LIN {X 0,Y 227.274,Z 763.314,A -85,B 0,C 180,E1 -20014.895,E2 -20014.895} C_VEL
LIN {X 0,Y 226.122,Z 765.679,A -85,B 0,C 180,E1 -20018.434,E2 -20018.434} C_VEL
LIN {X 0,Y 225.536,Z 766.463,A -85,B 0,C 180,E1 -20021.593,E2 -20021.593} C_VEL
LIN {X 0,Y 225.305,Z 766.2,A -85,B 0,C 180,E1 -20024.155,E2 -20024.155} C_VEL
LIN {X 0,Y 225.347,Z 765.158,A -85,B 0,C 180,E1 -20026.675,E2 -20026.675} C_VEL
LIN {X 0,Y 225.598,Z 763.327,A -85,B 0,C 180,E1 -20029.14,E2 -20029.14} C_VEL
LIN {X 0,Y 225.943,Z 760.772,A -85,B 0,C 180,E1 -20031.529,E2 -20031.529} C_VEL
LIN {X 0,Y 226.464,Z 757.485,A -85,B 0,C 180,E1 -20033.868,E2 -20033.868} C_VEL
LIN {X 0,Y 227.318,Z 752.537,A -85,B 0,C 180,E1 -20036.591,E2 -20036.591} C_VEL
LIN {X 0,Y 228.588,Z 745.96,A -85,B 0,C 180,E1 -20039.415,E2 -20039.415} C_VEL
LIN {X 0,Y 230.085,Z 738.559,A -85,B 0,C 180,E1 -20041.941,E2 -20041.941} C_VEL
LIN {X 0,Y 231.914,Z 729.456,A -85,B 0,C 180,E1 -20044.415,E2 -20044.415} C_VEL
LIN {X 0,Y 233.849,Z 719.737,A -85,B 0,C 180,E1 -20046.533,E2 -20046.533} C_VEL
LIN {X 0,Y 235.817,Z 708.858,A -85,B 0,C 180,E1 -20048.434,E2 -20048.434} C_VEL
LIN {X 0,Y 236.209,Z 705.915,A -85,B 0,C 180,E1 -20048.878,E2 -20048.878} C_VEL
LIN {X 0,Y 234.743,Z 695.22,A -85,B 0,C 180,E1 -20050.544,E2 -20050.544} C_VEL
LIN {X 0,Y 232.764,Z 684.343,A -85,B 0,C 180,E1 -20051.988,E2 -20051.988} C_VEL
LIN {X 0,Y 229.693,Z 671.184,A -85,B 0,C 180,E1 -20053.426,E2 -20053.426} C_VEL
LIN {X 0,Y 227.253,Z 661.617,A -85,B 0,C 180,E1 -20054.299,E2 -20054.299} C_VEL
LIN {X 0,Y 227.825,Z 657.568,A -85,B 0,C 180,E1 -20059.333,E2 -20059.333} C_VEL
LIN {X 0,Y 228.196,Z 656.059,A -85,B 0,C 180,E1 -20061.364,E2 -20061.364} C_VEL
LIN {X 0,Y 228.175,Z 656.064,A -85,B 0,C 180,E1 -20064.697,E2 -20064.697} C_VEL
LIN {X 0,Y 228.557,Z 656.012,A -85,B 0,C 180,E1 -20068.237,E2 -20068.237} C_VEL
LIN {X 0,Y 228.556,Z 656.01,A -85,B 0,C 180,E1 -20071.761,E2 -20071.761} C_VEL
LIN {X 0,Y 228.191,Z 656.057,A -85,B 0,C 180,E1 -20077.076,E2 -20077.076} C_VEL
LIN {X 0,Y 227.745,Z 656.119,A -85,B 0,C 180,E1 -20081.119,E2 -20081.119} C_VEL
LIN {X 0,Y 227.625,Z 656.245,A -85,B 0,C 180,E1 -20081.576,E2 -20081.576} C_VEL
LIN {X 0,Y 227.143,Z 659.782,A -85,B 0,C 180,E1 -20084.788,E2 -20084.788} C_VEL
LIN {X 0,Y 230.876,Z 674.703,A -85,B 0,C 180,E1 -20086.162,E2 -20086.162} C_VEL
LIN {X 0,Y 233.355,Z 686.703,A -85,B 0,C 180,E1 -20087.527,E2 -20087.527} C_VEL
LIN {X 0,Y 235.304,Z 698.674,A -85,B 0,C 180,E1 -20089.18,E2 -20089.18} C_VEL
LIN {X 0,Y 236.095,Z 705.463,A -85,B 0,C 180,E1 -20090.245,E2 -20090.245} C_VEL
LIN {X 0,Y 234.36,Z 715.909,A -85,B 0,C 180,E1 -20091.953,E2 -20091.953} C_VEL
LIN {X 0,Y 232.354,Z 726.447,A -85,B 0,C 180,E1 -20094.099,E2 -20094.099} C_VEL
LIN {X 0,Y 230.69,Z 734.831,A -85,B 0,C 180,E1 -20096.214,E2 -20096.214} C_VEL
LIN {X 0,Y 228.896,Z 743.456,A -85,B 0,C 180,E1 -20098.94,E2 -20098.94} C_VEL
LIN {X 0,Y 227.645,Z 750.251,A -85,B 0,C 180,E1 -20101.656,E2 -20101.656} C_VEL
LIN {X 0,Y 226.787,Z 754.751,A -85,B 0,C 180,E1 -20103.903,E2 -20103.903} C_VEL
LIN {X 0,Y 226.156,Z 758.446,A -85,B 0,C 180,E1 -20106.187,E2 -20106.187} C_VEL
LIN {X 0,Y 225.597,Z 761.739,A -85,B 0,C 180,E1 -20108.847,E2 -20108.847} C_VEL
LIN {X 0,Y 225.241,Z 764.045,A -85,B 0,C 180,E1 -20111.509,E2 -20111.509} C_VEL
LIN {X 0,Y 225.231,Z 765.419,A -85,B 0,C 180,E1 -20114.136,E2 -20114.136} C_VEL
LIN {X 0,Y 225.354,Z 765.922,A -85,B 0,C 180,E1 -20116.677,E2 -20116.677} C_VEL
LIN {X 0,Y 225.717,Z 765.607,A -85,B 0,C 180,E1 -20119.166,E2 -20119.166} C_VEL
LIN {X 0,Y 226.268,Z 764.569,A -85,B 0,C 180,E1 -20121.595,E2 -20121.595} C_VEL
LIN {X 0,Y 227.147,Z 762.813,A -85,B 0,C 180,E1 -20123.994,E2 -20123.994} C_VEL
LIN {X 0,Y 228.834,Z 758.808,A -85,B 0,C 180,E1 -20127.489,E2 -20127.489} C_VEL
LIN {X 0,Y 230.384,Z 754.929,A -85,B 0,C 180,E1 -20129.916,E2 -20129.916} C_VEL
LIN {X 0,Y 232.388,Z 749.966,A -85,B 0,C 180,E1 -20132.35,E2 -20132.35} C_VEL
LIN {X 0,Y 234.755,Z 743.842,A -85,B 0,C 180,E1 -20134.744,E2 -20134.744} C_VEL
LIN {X 0,Y 237.51,Z 736.342,A -85,B 0,C 180,E1 -20137.093,E2 -20137.093} C_VEL
LIN {X 0,Y 240.476,Z 727.629,A -85,B 0,C 180,E1 -20139.26,E2 -20139.26} C_VEL
LIN {X 0,Y 243.611,Z 717.397,A -85,B 0,C 180,E1 -20141.28,E2 -20141.28} C_VEL
LIN {X 0,Y 244.299,Z 713.897,A -85,B 0,C 180,E1 -20141.926,E2 -20141.926} C_VEL
LIN {X 0,Y 243.791,Z 704.371,A -85,B 0,C 180,E1 -20143.891,E2 -20143.891} C_VEL
LIN {X 0,Y 242.005,Z 693.516,A -85,B 0,C 180,E1 -20146.031,E2 -20146.031} C_VEL
LIN {X 0,Y 239.114,Z 682.956,A -85,B 0,C 180,E1 -20148.127,E2 -20148.127} C_VEL
LIN {X 0,Y 235.916,Z 674.484,A -85,B 0,C 180,E1 -20149.85,E2 -20149.85} C_VEL
LIN {X 0,Y 233.629,Z 669.665,A -85,B 0,C 180,E1 -20150.93,E2 -20150.93} C_VEL
LIN {X 0,Y 231.756,Z 665.99,A -85,B 0,C 180,E1 -20151.773,E2 -20151.773} C_VEL
LIN {X 0,Y 229.771,Z 662.892,A -85,B 0,C 180,E1 -20152.586,E2 -20152.586} C_VEL
LIN {X 0,Y 229.263,Z 661.334,A -85,B 0,C 180,E1 -20152.901,E2 -20152.901} C_VEL
LIN {X 0,Y 228.776,Z 657.181,A -85,B 0,C 180,E1 -20158.24,E2 -20158.24} C_VEL
LIN {X 0,Y 228.623,Z 656.007,A -85,B 0,C 180,E1 -20160,E2 -20160} C_VEL
LIN {X 0,Y 228.553,Z 656.016,A -85,B 0,C 180,E1 -20161.762,E2 -20161.762} C_VEL
LIN {X 0,Y 228.355,Z 656.04,A -85,B 0,C 180,E1 -20167.071,E2 -20167.071} C_VEL
LIN {X 0,Y 228.169,Z 656.065,A -85,B 0,C 180,E1 -20170.65,E2 -20170.65} C_VEL
LIN {X 0,Y 228.055,Z 656.076,A -85,B 0,C 180,E1 -20176.102,E2 -20176.102} C_VEL
LIN {X 0,Y 227.94,Z 656.092,A -85,B 0,C 180,E1 -20179.826,E2 -20179.826} C_VEL
LIN {X 0,Y 227.911,Z 656.092,A -85,B 0,C 180,E1 -20183.633,E2 -20183.633} C_VEL
LIN {X 0,Y 227.883,Z 656.1,A -85,B 0,C 180,E1 -20187.555,E2 -20187.555} C_VEL
LIN {X 0,Y 227.869,Z 656.1,A -85,B 0,C 180,E1 -20191.622,E2 -20191.622} C_VEL
LIN {X 0,Y 227.88,Z 656.097,A -85,B 0,C 180,E1 -20195.872,E2 -20195.872} C_VEL
LIN {X 0,Y 227.829,Z 656.101,A -85,B 0,C 180,E1 -20198.548,E2 -20198.548} C_VEL
LIN {X 0,Y 227.18,Z 656.345,A -85,B 0,C 180,E1 -20200.022,E2 -20200.022} C_VEL
LIN {X 0,Y 225.688,Z 657.012,A -85,B 0,C 180,E1 -20201.468,E2 -20201.468} C_VEL
LIN {X 0,Y 222.387,Z 659.357,A -85,B 0,C 180,E1 -20204.352,E2 -20204.352} C_VEL
LIN {X 0,Y 221.675,Z 660.931,A -85,B 0,C 180,E1 -20205.825,E2 -20205.825} C_VEL
LIN {X 0,Y 221.72,Z 661.5,A -85,B 0,C 180,E1 -20206.317,E2 -20206.317} C_VEL
LIN {X 0,Y 222.548,Z 665.01,A -85,B 0,C 180,E1 -20209.016,E2 -20209.016} C_VEL
LIN {X 0,Y 225.07,Z 669.34,A -85,B 0,C 180,E1 -20210.166,E2 -20210.166} C_VEL
LIN {X 0,Y 226.351,Z 672.017,A -85,B 0,C 180,E1 -20210.777,E2 -20210.777} C_VEL
LIN {X 0,Y 228.189,Z 675.676,A -85,B 0,C 180,E1 -20211.635,E2 -20211.635} C_VEL
LIN {X 0,Y 231.062,Z 684.216,A -85,B 0,C 180,E1 -20213.274,E2 -20213.274} C_VEL
LIN {X 0,Y 233.784,Z 695.583,A -85,B 0,C 180,E1 -20215.343,E2 -20215.343} C_VEL
LIN {X 0,Y 235.256,Z 705.746,A -85,B 0,C 180,E1 -20217.171,E2 -20217.171} C_VEL
LIN {X 0,Y 235.869,Z 716.507,A -85,B 0,C 180,E1 -20219.195,E2 -20219.195} C_VEL
LIN {X 0,Y 235.472,Z 726.605,A -85,B 0,C 180,E1 -20221.221,E2 -20221.221} C_VEL
LIN {X 0,Y 234.448,Z 733.894,A -85,B 0,C 180,E1 -20222.798,E2 -20222.798} C_VEL
LIN {X 0,Y 231.402,Z 742.92,A -85,B 0,C 180,E1 -20224.838,E2 -20224.838} C_VEL
LIN {X 0,Y 228.129,Z 751.752,A -85,B 0,C 180,E1 -20227.353,E2 -20227.353} C_VEL
LIN {X 0,Y 225.399,Z 758.948,A -85,B 0,C 180,E1 -20229.942,E2 -20229.942} C_VEL
LIN {X 0,Y 223.2,Z 764.764,A -85,B 0,C 180,E1 -20232.595,E2 -20232.595} C_VEL
LIN {X 0,Y 221.234,Z 769.387,A -85,B 0,C 180,E1 -20235.278,E2 -20235.278} C_VEL
LIN {X 0,Y 219.983,Z 772.932,A -85,B 0,C 180,E1 -20238.016,E2 -20238.016} C_VEL
LIN {X 0,Y 219.133,Z 775.505,A -85,B 0,C 180,E1 -20240.773,E2 -20240.773} C_VEL
LIN {X 0,Y 218.765,Z 776.719,A -85,B 0,C 180,E1 -20242.618,E2 -20242.618} C_VEL
LIN {X 0,Y 218.557,Z 777.78,A -85,B 0,C 180,E1 -20245.45,E2 -20245.45} C_VEL
LIN {X 0,Y 218.602,Z 778.042,A -85,B 0,C 180,E1 -20248.158,E2 -20248.158} C_VEL
LIN {X 0,Y 218.67,Z 778.897,A -85,B 0,C 180,E1 -20250.001,E2 -20250.001} C_VEL
LIN {X 0,Y 218.561,Z 779.313,A -85,B 0,C 180,E1 -20251.843,E2 -20251.843} C_VEL
LIN {X 0,Y 218.597,Z 778.94,A -85,B 0,C 180,E1 -20255.536,E2 -20255.536} C_VEL
LIN {X 0,Y 218.797,Z 778.178,A -85,B 0,C 180,E1 -20257.383,E2 -20257.383} C_VEL
LIN {X 0,Y 219.145,Z 777.013,A -85,B 0,C 180,E1 -20259.228,E2 -20259.228} C_VEL
LIN {X 0,Y 220.412,Z 773.422,A -85,B 0,C 180,E1 -20262.898,E2 -20262.898} C_VEL
LIN {X 0,Y 221.86,Z 769.607,A -85,B 0,C 180,E1 -20265.621,E2 -20265.621} C_VEL
LIN {X 0,Y 223.99,Z 764.713,A -85,B 0,C 180,E1 -20268.287,E2 -20268.287} C_VEL
LIN {X 0,Y 226.381,Z 758.62,A -85,B 0,C 180,E1 -20270.918,E2 -20270.918} C_VEL
LIN {X 0,Y 229.184,Z 751.13,A -85,B 0,C 180,E1 -20273.494,E2 -20273.494} C_VEL
LIN {X 0,Y 232.086,Z 743.584,A -85,B 0,C 180,E1 -20275.564,E2 -20275.564} C_VEL
LIN {X 0,Y 235.421,Z 733.539,A -85,B 0,C 180,E1 -20277.805,E2 -20277.805} C_VEL
LIN {X 0,Y 236.271,Z 724.664,A -85,B 0,C 180,E1 -20279.735,E2 -20279.735} C_VEL
LIN {X 0,Y 236.179,Z 715.261,A -85,B 0,C 180,E1 -20281.657,E2 -20281.657} C_VEL
LIN {X 0,Y 235.121,Z 705.444,A -85,B 0,C 180,E1 -20283.616,E2 -20283.616} C_VEL
LIN {X 0,Y 233.152,Z 695.824,A -85,B 0,C 180,E1 -20285.524,E2 -20285.524} C_VEL
LIN {X 0,Y 229.982,Z 685.655,A -85,B 0,C 180,E1 -20287.675,E2 -20287.675} C_VEL
LIN {X 0,Y 228.05,Z 681.227,A -85,B 0,C 180,E1 -20288.719,E2 -20288.719} C_VEL
LIN {X 0,Y 226.282,Z 677.271,A -85,B 0,C 180,E1 -20289.681,E2 -20289.681} C_VEL
LIN {X 0,Y 223.674,Z 673.089,A -85,B 0,C 180,E1 -20290.949,E2 -20290.949} C_VEL
LIN {X 0,Y 223.107,Z 671.11,A -85,B 0,C 180,E1 -20291.351,E2 -20291.351} C_VEL
LIN {X 0,Y 222.919,Z 669.385,A -85,B 0,C 180,E1 -20293.916,E2 -20293.916} C_VEL
LIN {X 0,Y 222.468,Z 666.7,A -85,B 0,C 180,E1 -20298.439,E2 -20298.439} C_VEL
LIN {X 0,Y 222.139,Z 664.407,A -85,B 0,C 180,E1 -20303.05,E2 -20303.05} C_VEL
LIN {X 0,Y 221.847,Z 662.686,A -85,B 0,C 180,E1 -20307.415,E2 -20307.415} C_VEL
LIN {X 0,Y 221.656,Z 661.448,A -85,B 0,C 180,E1 -20311.601,E2 -20311.601} C_VEL
LIN {X 0,Y 221.53,Z 660.632,A -85,B 0,C 180,E1 -20315.643,E2 -20315.643} C_VEL
LIN {X 0,Y 221.475,Z 660.194,A -85,B 0,C 180,E1 -20319.57,E2 -20319.57} C_VEL
LIN {X 0,Y 221.582,Z 660.074,A -85,B 0,C 180,E1 -20323.414,E2 -20323.414} C_VEL
LIN {X 0,Y 221.654,Z 660.293,A -85,B 0,C 180,E1 -20327.176,E2 -20327.176} C_VEL
LIN {X 0,Y 221.899,Z 660.774,A -85,B 0,C 180,E1 -20330.888,E2 -20330.888} C_VEL
LIN {X 0,Y 222.014,Z 661.565,A -85,B 0,C 180,E1 -20334.551,E2 -20334.551} C_VEL
LIN {X 0,Y 222.44,Z 662.548,A -85,B 0,C 180,E1 -20338.19,E2 -20338.19} C_VEL
LIN {X 0,Y 222.644,Z 663.12,A -85,B 0,C 180,E1 -20340,E2 -20340} C_VEL
LIN {X 0,Y 222.533,Z 664.557,A -85,B 0,C 180,E1 -20343.565,E2 -20343.565} C_VEL
LIN {X 0,Y 223.667,Z 667.608,A -85,B 0,C 180,E1 -20344.281,E2 -20344.281} C_VEL
LIN {X 0,Y 225.776,Z 670.33,A -85,B 0,C 180,E1 -20345.268,E2 -20345.268} C_VEL
LIN {X 0,Y 227.849,Z 674.14,A -85,B 0,C 180,E1 -20346.364,E2 -20346.364} C_VEL
LIN {X 0,Y 231.352,Z 681.619,A -85,B 0,C 180,E1 -20348.297,E2 -20348.297} C_VEL
LIN {X 0,Y 234.93,Z 692.21,A -85,B 0,C 180,E1 -20350.775,E2 -20350.775} C_VEL
LIN {X 0,Y 237.082,Z 701.465,A -85,B 0,C 180,E1 -20352.846,E2 -20352.846} C_VEL
LIN {X 0,Y 238.267,Z 710.869,A -85,B 0,C 180,E1 -20354.957,E2 -20354.957} C_VEL
LIN {X 0,Y 238.439,Z 717.51,A -85,B 0,C 180,E1 -20356.481,E2 -20356.481} C_VEL
LIN {X 0,Y 235.322,Z 727.408,A -85,B 0,C 180,E1 -20358.464,E2 -20358.464} C_VEL
LIN {X 0,Y 232.446,Z 735.279,A -85,B 0,C 180,E1 -20360.398,E2 -20360.398} C_VEL
LIN {X 0,Y 229.065,Z 743.764,A -85,B 0,C 180,E1 -20363.009,E2 -20363.009} C_VEL
LIN {X 0,Y 226.156,Z 750.779,A -85,B 0,C 180,E1 -20365.789,E2 -20365.789} C_VEL
LIN {X 0,Y 223.837,Z 756.029,A -85,B 0,C 180,E1 -20368.46,E2 -20368.46} C_VEL
LIN {X 0,Y 221.945,Z 760.206,A -85,B 0,C 180,E1 -20371.243,E2 -20371.243} C_VEL
LIN {X 0,Y 220.515,Z 763.269,A -85,B 0,C 180,E1 -20374.04,E2 -20374.04} C_VEL
LIN {X 0,Y 219.266,Z 765.708,A -85,B 0,C 180,E1 -20377.517,E2 -20377.517} C_VEL
LIN {X 0,Y 218.668,Z 766.536,A -85,B 0,C 180,E1 -20380.001,E2 -20380.001} C_VEL
LIN {X 0,Y 218.324,Z 766.658,A -85,B 0,C 180,E1 -20382.532,E2 -20382.532} C_VEL
LIN {X 0,Y 218.212,Z 766.033,A -85,B 0,C 180,E1 -20385.118,E2 -20385.118} C_VEL
LIN {X 0,Y 218.347,Z 764.572,A -85,B 0,C 180,E1 -20387.758,E2 -20387.758} C_VEL
LIN {X 0,Y 218.651,Z 762.155,A -85,B 0,C 180,E1 -20390.482,E2 -20390.482} C_VEL
LIN {X 0,Y 219.182,Z 758.661,A -85,B 0,C 180,E1 -20393.285,E2 -20393.285} C_VEL
LIN {X 0,Y 220.04,Z 753.926,A -85,B 0,C 180,E1 -20396.143,E2 -20396.143} C_VEL
LIN {X 0,Y 221.243,Z 747.658,A -85,B 0,C 180,E1 -20399.058,E2 -20399.058} C_VEL
LIN {X 0,Y 222.923,Z 739.639,A -85,B 0,C 180,E1 -20401.976,E2 -20401.976} C_VEL
LIN {X 0,Y 224.749,Z 730.916,A -85,B 0,C 180,E1 -20404.5,E2 -20404.5} C_VEL
LIN {X 0,Y 226.878,Z 720.727,A -85,B 0,C 180,E1 -20406.83,E2 -20406.83} C_VEL
LIN {X 0,Y 228.961,Z 709.618,A -85,B 0,C 180,E1 -20408.858,E2 -20408.858} C_VEL
LIN {X 0,Y 229.303,Z 706.457,A -85,B 0,C 180,E1 -20409.361,E2 -20409.361} C_VEL
LIN {X 0,Y 227.826,Z 695.656,A -85,B 0,C 180,E1 -20411.1,E2 -20411.1} C_VEL
LIN {X 0,Y 225.656,Z 683.949,A -85,B 0,C 180,E1 -20412.7,E2 -20412.7} C_VEL
LIN {X 0,Y 222.676,Z 671.185,A -85,B 0,C 180,E1 -20414.144,E2 -20414.144} C_VEL
LIN {X 0,Y 220.233,Z 661.821,A -85,B 0,C 180,E1 -20415.031,E2 -20415.031} C_VEL
LIN {X 0,Y 221.106,Z 657.109,A -85,B 0,C 180,E1 -20421.085,E2 -20421.085} C_VEL
LIN {X 0,Y 221.219,Z 656.926,A -85,B 0,C 180,E1 -20422.699,E2 -20422.699} C_VEL
LIN {X 0,Y 221.515,Z 656.889,A -85,B 0,C 180,E1 -20428.181,E2 -20428.181} C_VEL
LIN {X 0,Y 221.514,Z 656.887,A -85,B 0,C 180,E1 -20431.817,E2 -20431.817} C_VEL
LIN {X 0,Y 221.117,Z 656.936,A -85,B 0,C 180,E1 -20437.303,E2 -20437.303} C_VEL
LIN {X 0,Y 220.707,Z 656.995,A -85,B 0,C 180,E1 -20441.014,E2 -20441.014} C_VEL
LIN {X 0,Y 220.6,Z 657.157,A -85,B 0,C 180,E1 -20441.484,E2 -20441.484} C_VEL
LIN {X 0,Y 220.152,Z 660.141,A -85,B 0,C 180,E1 -20444.087,E2 -20444.087} C_VEL
LIN {X 0,Y 223.775,Z 674.308,A -85,B 0,C 180,E1 -20445.424,E2 -20445.424} C_VEL
LIN {X 0,Y 226.417,Z 686.993,A -85,B 0,C 180,E1 -20446.917,E2 -20446.917} C_VEL
LIN {X 0,Y 228.362,Z 698.959,A -85,B 0,C 180,E1 -20448.62,E2 -20448.62} C_VEL
LIN {X 0,Y 229.151,Z 707.109,A -85,B 0,C 180,E1 -20449.949,E2 -20449.949} C_VEL
LIN {X 0,Y 227,Z 718.98,A -85,B 0,C 180,E1 -20452.023,E2 -20452.023} C_VEL
LIN {X 0,Y 224.908,Z 729.43,A -85,B 0,C 180,E1 -20454.366,E2 -20454.366} C_VEL
LIN {X 0,Y 223.155,Z 737.692,A -85,B 0,C 180,E1 -20456.665,E2 -20456.665} C_VEL
LIN {X 0,Y 221.495,Z 745.734,A -85,B 0,C 180,E1 -20459.459,E2 -20459.459} C_VEL
LIN {X 0,Y 220.225,Z 752.202,A -85,B 0,C 180,E1 -20462.329,E2 -20462.329} C_VEL
LIN {X 0,Y 219.303,Z 757.291,A -85,B 0,C 180,E1 -20465.228,E2 -20465.228} C_VEL
LIN {X 0,Y 218.712,Z 760.533,A -85,B 0,C 180,E1 -20467.627,E2 -20467.627} C_VEL
LIN {X 0,Y 218.292,Z 763.053,A -85,B 0,C 180,E1 -20470.082,E2 -20470.082} C_VEL
LIN {X 0,Y 218.126,Z 764.828,A -85,B 0,C 180,E1 -20472.579,E2 -20472.579} C_VEL
LIN {X 0,Y 218.143,Z 765.841,A -85,B 0,C 180,E1 -20475.135,E2 -20475.135} C_VEL
LIN {X 0,Y 218.379,Z 766.099,A -85,B 0,C 180,E1 -20477.747,E2 -20477.747} C_VEL
LIN {X 0,Y 218.862,Z 765.548,A -85,B 0,C 180,E1 -20480.413,E2 -20480.413} C_VEL
LIN {X 0,Y 219.68,Z 764.139,A -85,B 0,C 180,E1 -20483.109,E2 -20483.109} C_VEL
LIN {X 0,Y 220.824,Z 761.805,A -85,B 0,C 180,E1 -20485.839,E2 -20485.839} C_VEL
LIN {X 0,Y 222.359,Z 758.453,A -85,B 0,C 180,E1 -20488.579,E2 -20488.579} C_VEL
LIN {X 0,Y 224.29,Z 753.948,A -85,B 0,C 180,E1 -20491.324,E2 -20491.324} C_VEL
LIN {X 0,Y 227.066,Z 747.424,A -85,B 0,C 180,E1 -20494.321,E2 -20494.321} C_VEL
LIN {X 0,Y 229.652,Z 740.988,A -85,B 0,C 180,E1 -20496.645,E2 -20496.645} C_VEL
LIN {X 0,Y 233.016,Z 732.041,A -85,B 0,C 180,E1 -20499.224,E2 -20499.224} C_VEL
LIN {X 0,Y 236.323,Z 722.47,A -85,B 0,C 180,E1 -20501.367,E2 -20501.367} C_VEL
LIN {X 0,Y 238.115,Z 716.596,A -85,B 0,C 180,E1 -20502.479,E2 -20502.479} C_VEL
LIN {X 0,Y 238.001,Z 708.977,A -85,B 0,C 180,E1 -20504.148,E2 -20504.148} C_VEL
LIN {X 0,Y 236.866,Z 699.006,A -85,B 0,C 180,E1 -20506.269,E2 -20506.269} C_VEL
LIN {X 0,Y 234.397,Z 688.259,A -85,B 0,C 180,E1 -20508.549,E2 -20508.549} C_VEL
LIN {X 0,Y 231.629,Z 679.76,A -85,B 0,C 180,E1 -20510.393,E2 -20510.393} C_VEL
LIN {X 0,Y 227.968,Z 671.519,A -85,B 0,C 180,E1 -20512.36,E2 -20512.36} C_VEL
LIN {X 0,Y 225.794,Z 667.824,A -85,B 0,C 180,E1 -20513.403,E2 -20513.403} C_VEL
LIN {X 0,Y 225.19,Z 666.7,A -85,B 0,C 180,E1 -20513.701,E2 -20513.701} C_VEL
LIN {X 0,Y 222.867,Z 663.564,A -85,B 0,C 180,E1 -20514.742,E2 -20514.742} C_VEL
LIN {X 0,Y 222.097,Z 661.579,A -85,B 0,C 180,E1 -20515.235,E2 -20515.235} C_VEL
LIN {X 0,Y 222.014,Z 659.376,A -85,B 0,C 180,E1 -20518.186,E2 -20518.186} C_VEL
LIN {X 0,Y 221.861,Z 658.117,A -85,B 0,C 180,E1 -20520,E2 -20520} C_VEL
LIN {X 0,Y 221.411,Z 656.905,A -85,B 0,C 180,E1 -20522.274,E2 -20522.274} C_VEL
LIN {X 0,Y 221.292,Z 656.918,A -85,B 0,C 180,E1 -20527.298,E2 -20527.298} C_VEL
LIN {X 0,Y 221.114,Z 656.943,A -85,B 0,C 180,E1 -20530.994,E2 -20530.994} C_VEL
LIN {X 0,Y 221.014,Z 656.952,A -85,B 0,C 180,E1 -20536.63,E2 -20536.63} C_VEL
LIN {X 0,Y 220.89,Z 656.97,A -85,B 0,C 180,E1 -20540.486,E2 -20540.486} C_VEL
LIN {X 0,Y 220.865,Z 656.971,A -85,B 0,C 180,E1 -20544.435,E2 -20544.435} C_VEL
LIN {X 0,Y 220.833,Z 656.974,A -85,B 0,C 180,E1 -20548.514,E2 -20548.514} C_VEL
LIN {X 0,Y 220.817,Z 656.977,A -85,B 0,C 180,E1 -20552.756,E2 -20552.756} C_VEL
LIN {X 0,Y 220.808,Z 656.978,A -85,B 0,C 180,E1 -20557.279,E2 -20557.279} C_VEL
LIN {X 0,Y 220.841,Z 657.097,A -85,B 0,C 180,E1 -20562.075,E2 -20562.075} C_VEL
LIN {X 0,Y 221.72,Z 661.5,A -85,B 0,C 180,E1 -20566.317,E2 -20566.317} C_VEL
LIN {X 0,Y 221.973,Z 663.118,A -85,B 0,C 180,E1 -20567.228,E2 -20567.228} C_VEL
LIN {X 0,Y 222.349,Z 666.854,A -85,B 0,C 180,E1 -20568.397,E2 -20568.397} C_VEL
LIN {X 0,Y 222.787,Z 671.469,A -85,B 0,C 180,E1 -20569.362,E2 -20569.362} C_VEL
LIN {X 0,Y 224.433,Z 681.719,A -85,B 0,C 180,E1 -20571.11,E2 -20571.11} C_VEL
LIN {X 0,Y 225.374,Z 684.864,A -85,B 0,C 180,E1 -20571.747,E2 -20571.747} C_VEL
LIN {X 0,Y 228.202,Z 697.223,A -85,B 0,C 180,E1 -20574.188,E2 -20574.188} C_VEL
LIN {X 0,Y 229.505,Z 707.571,A -85,B 0,C 180,E1 -20576.198,E2 -20576.198} C_VEL
LIN {X 0,Y 229.903,Z 718.016,A -85,B 0,C 180,E1 -20578.284,E2 -20578.284} C_VEL
LIN {X 0,Y 229.312,Z 727.779,A -85,B 0,C 180,E1 -20580.367,E2 -20580.367} C_VEL
LIN {X 0,Y 228.204,Z 734.892,A -85,B 0,C 180,E1 -20581.989,E2 -20581.989} C_VEL
LIN {X 0,Y 224.465,Z 745.253,A -85,B 0,C 180,E1 -20584.501,E2 -20584.501} C_VEL
LIN {X 0,Y 221.086,Z 753.621,A -85,B 0,C 180,E1 -20587.083,E2 -20587.083} C_VEL
LIN {X 0,Y 218.368,Z 760.368,A -85,B 0,C 180,E1 -20589.759,E2 -20589.759} C_VEL
LIN {X 0,Y 215.698,Z 766.649,A -85,B 0,C 180,E1 -20592.949,E2 -20592.949} C_VEL
LIN {X 0,Y 213.874,Z 770.799,A -85,B 0,C 180,E1 -20595.733,E2 -20595.733} C_VEL
LIN {X 0,Y 212.678,Z 773.917,A -85,B 0,C 180,E1 -20598.565,E2 -20598.565} C_VEL
LIN {X 0,Y 212.102,Z 775.49,A -85,B 0,C 180,E1 -20600.464,E2 -20600.464} C_VEL
LIN {X 0,Y 211.506,Z 777.357,A -85,B 0,C 180,E1 -20604.28,E2 -20604.28} C_VEL
LIN {X 0,Y 211.518,Z 777.685,A -85,B 0,C 180,E1 -20608.097,E2 -20608.097} C_VEL
LIN {X 0,Y 211.584,Z 778.581,A -85,B 0,C 180,E1 -20610.001,E2 -20610.001} C_VEL
LIN {X 0,Y 211.46,Z 779.069,A -85,B 0,C 180,E1 -20611.905,E2 -20611.905} C_VEL
LIN {X 0,Y 211.42,Z 779.072,A -85,B 0,C 180,E1 -20614.242,E2 -20614.242} C_VEL
LIN {X 0,Y 211.727,Z 778.068,A -85,B 0,C 180,E1 -20617.631,E2 -20617.631} C_VEL
LIN {X 0,Y 212.113,Z 776.971,A -85,B 0,C 180,E1 -20619.537,E2 -20619.537} C_VEL
LIN {X 0,Y 212.698,Z 775.45,A -85,B 0,C 180,E1 -20621.436,E2 -20621.436} C_VEL
LIN {X 0,Y 213.924,Z 772.4,A -85,B 0,C 180,E1 -20624.265,E2 -20624.265} C_VEL
LIN {X 0,Y 215.753,Z 768.336,A -85,B 0,C 180,E1 -20627.048,E2 -20627.048} C_VEL
LIN {X 0,Y 218.134,Z 763.17,A -85,B 0,C 180,E1 -20629.774,E2 -20629.774} C_VEL
LIN {X 0,Y 221.044,Z 755.95,A -85,B 0,C 180,E1 -20632.773,E2 -20632.773} C_VEL
LIN {X 0,Y 223.877,Z 748.942,A -85,B 0,C 180,E1 -20635.075,E2 -20635.075} C_VEL
LIN {X 0,Y 227.661,Z 739.285,A -85,B 0,C 180,E1 -20637.585,E2 -20637.585} C_VEL
LIN {X 0,Y 229.012,Z 735.538,A -85,B 0,C 180,E1 -20638.404,E2 -20638.404} C_VEL
LIN {X 0,Y 230.059,Z 727.441,A -85,B 0,C 180,E1 -20640.279,E2 -20640.279} C_VEL
LIN {X 0,Y 230.291,Z 717.897,A -85,B 0,C 180,E1 -20642.378,E2 -20642.378} C_VEL
LIN {X 0,Y 229.457,Z 708.099,A -85,B 0,C 180,E1 -20644.464,E2 -20644.464} C_VEL
LIN {X 0,Y 227.644,Z 698.143,A -85,B 0,C 180,E1 -20646.612,E2 -20646.612} C_VEL
LIN {X 0,Y 224.992,Z 689.26,A -85,B 0,C 180,E1 -20648.663,E2 -20648.663} C_VEL
LIN {X 0,Y 221.766,Z 681.602,A -85,B 0,C 180,E1 -20650.686,E2 -20650.686} C_VEL
LIN {X 0,Y 219.7,Z 677.836,A -85,B 0,C 180,E1 -20651.848,E2 -20651.848} C_VEL
LIN {X 0,Y 219.151,Z 676.556,A -85,B 0,C 180,E1 -20652.189,E2 -20652.189} C_VEL
LIN {X 0,Y 216.932,Z 673.503,A -85,B 0,C 180,E1 -20653.396,E2 -20653.396} C_VEL
LIN {X 0,Y 215.932,Z 670.691,A -85,B 0,C 180,E1 -20654.148,E2 -20654.148} C_VEL
LIN {X 0,Y 215.521,Z 668.156,A -85,B 0,C 180,E1 -20658.593,E2 -20658.593} C_VEL
LIN {X 0,Y 215.296,Z 666.644,A -85,B 0,C 180,E1 -20661.667,E2 -20661.667} C_VEL
LIN {X 0,Y 214.986,Z 664.771,A -85,B 0,C 180,E1 -20666.238,E2 -20666.238} C_VEL
LIN {X 0,Y 214.788,Z 663.394,A -85,B 0,C 180,E1 -20670.606,E2 -20670.606} C_VEL
LIN {X 0,Y 214.672,Z 662.477,A -85,B 0,C 180,E1 -20674.812,E2 -20674.812} C_VEL
LIN {X 0,Y 214.595,Z 661.963,A -85,B 0,C 180,E1 -20678.884,E2 -20678.884} C_VEL
LIN {X 0,Y 214.673,Z 661.783,A -85,B 0,C 180,E1 -20682.864,E2 -20682.864} C_VEL
LIN {X 0,Y 214.754,Z 661.943,A -85,B 0,C 180,E1 -20686.757,E2 -20686.757} C_VEL
LIN {X 0,Y 214.976,Z 662.379,A -85,B 0,C 180,E1 -20690.592,E2 -20690.592} C_VEL
LIN {X 0,Y 215.107,Z 663.127,A -85,B 0,C 180,E1 -20694.375,E2 -20694.375} C_VEL
LIN {X 0,Y 215.498,Z 664.087,A -85,B 0,C 180,E1 -20698.131,E2 -20698.131} C_VEL
LIN {X 0,Y 215.695,Z 665.116,A -85,B 0,C 180,E1 -20700.934,E2 -20700.934} C_VEL
LIN {X 0,Y 216.682,Z 667.712,A -85,B 0,C 180,E1 -20701.626,E2 -20701.626} C_VEL
LIN {X 0,Y 219.132,Z 670.979,A -85,B 0,C 180,E1 -20702.982,E2 -20702.982} C_VEL
LIN {X 0,Y 220.961,Z 674.492,A -85,B 0,C 180,E1 -20704.104,E2 -20704.104} C_VEL
LIN {X 0,Y 221.835,Z 675.57,A -85,B 0,C 180,E1 -20704.543,E2 -20704.543} C_VEL
LIN {X 0,Y 225.531,Z 683.247,A -85,B 0,C 180,E1 -20706.823,E2 -20706.823} C_VEL
LIN {X 0,Y 228.825,Z 692.912,A -85,B 0,C 180,E1 -20709.297,E2 -20709.297} C_VEL
LIN {X 0,Y 230.898,Z 701.564,A -85,B 0,C 180,E1 -20711.411,E2 -20711.411} C_VEL
LIN {X 0,Y 232.133,Z 710.583,A -85,B 0,C 180,E1 -20713.57,E2 -20713.57} C_VEL
LIN {X 0,Y 232.377,Z 717.84,A -85,B 0,C 180,E1 -20715.345,E2 -20715.345} C_VEL
LIN {X 0,Y 232.206,Z 719.832,A -85,B 0,C 180,E1 -20715.807,E2 -20715.807} C_VEL
LIN {X 0,Y 228.771,Z 729.635,A -85,B 0,C 180,E1 -20717.891,E2 -20717.891} C_VEL
LIN {X 0,Y 225.013,Z 739.102,A -85,B 0,C 180,E1 -20720.443,E2 -20720.443} C_VEL
LIN {X 0,Y 221.649,Z 746.885,A -85,B 0,C 180,E1 -20723.142,E2 -20723.142} C_VEL
LIN {X 0,Y 218.813,Z 753.095,A -85,B 0,C 180,E1 -20725.93,E2 -20725.93} C_VEL
LIN {X 0,Y 216.132,Z 758.636,A -85,B 0,C 180,E1 -20729.194,E2 -20729.194} C_VEL
LIN {X 0,Y 213.971,Z 762.957,A -85,B 0,C 180,E1 -20732.816,E2 -20732.816} C_VEL
LIN {X 0,Y 212.447,Z 765.693,A -85,B 0,C 180,E1 -20736.546,E2 -20736.546} C_VEL
LIN {X 0,Y 211.546,Z 766.871,A -85,B 0,C 180,E1 -20740.171,E2 -20740.171} C_VEL
LIN {X 0,Y 211.183,Z 766.798,A -85,B 0,C 180,E1 -20742.933,E2 -20742.933} C_VEL
LIN {X 0,Y 211.11,Z 765.91,A -85,B 0,C 180,E1 -20745.644,E2 -20745.644} C_VEL
LIN {X 0,Y 211.3,Z 764.262,A -85,B 0,C 180,E1 -20748.3,E2 -20748.3} C_VEL
LIN {X 0,Y 211.807,Z 760.75,A -85,B 0,C 180,E1 -20751.877,E2 -20751.877} C_VEL
LIN {X 0,Y 212.466,Z 756.965,A -85,B 0,C 180,E1 -20754.598,E2 -20754.598} C_VEL
LIN {X 0,Y 213.481,Z 751.453,A -85,B 0,C 180,E1 -20757.658,E2 -20757.658} C_VEL
LIN {X 0,Y 214.943,Z 744.515,A -85,B 0,C 180,E1 -20760.629,E2 -20760.629} C_VEL
LIN {X 0,Y 216.712,Z 736.274,A -85,B 0,C 180,E1 -20763.424,E2 -20763.424} C_VEL
LIN {X 0,Y 218.626,Z 727.54,A -85,B 0,C 180,E1 -20765.803,E2 -20765.803} C_VEL
LIN {X 0,Y 220.458,Z 718.556,A -85,B 0,C 180,E1 -20767.792,E2 -20767.792} C_VEL
LIN {X 0,Y 222.414,Z 708.097,A -85,B 0,C 180,E1 -20769.66,E2 -20769.66} C_VEL
LIN {X 0,Y 221.11,Z 697.449,A -85,B 0,C 180,E1 -20771.466,E2 -20771.466} C_VEL
LIN {X 0,Y 218.973,Z 685.436,A -85,B 0,C 180,E1 -20773.21,E2 -20773.21} C_VEL
LIN {X 0,Y 216.084,Z 672.839,A -85,B 0,C 180,E1 -20774.737,E2 -20774.737} C_VEL
LIN {X 0,Y 213.257,Z 662.022,A -85,B 0,C 180,E1 -20775.811,E2 -20775.811} C_VEL
LIN {X 0,Y 214.14,Z 657.81,A -85,B 0,C 180,E1 -20781.506,E2 -20781.506} C_VEL
LIN {X 0,Y 214.448,Z 657.769,A -85,B 0,C 180,E1 -20788.121,E2 -20788.121} C_VEL
LIN {X 0,Y 214.554,Z 657.758,A -85,B 0,C 180,E1 -20789.999,E2 -20789.999} C_VEL
LIN {X 0,Y 214.446,Z 657.767,A -85,B 0,C 180,E1 -20791.877,E2 -20791.877} C_VEL
LIN {X 0,Y 214.048,Z 657.816,A -85,B 0,C 180,E1 -20797.546,E2 -20797.546} C_VEL
LIN {X 0,Y 213.598,Z 657.881,A -85,B 0,C 180,E1 -20801.145,E2 -20801.145} C_VEL
LIN {X 0,Y 213.194,Z 660.098,A -85,B 0,C 180,E1 -20803.28,E2 -20803.28} C_VEL
LIN {X 0,Y 216.899,Z 674.695,A -85,B 0,C 180,E1 -20804.723,E2 -20804.723} C_VEL
LIN {X 0,Y 219.508,Z 687.258,A -85,B 0,C 180,E1 -20806.268,E2 -20806.268} C_VEL
LIN {X 0,Y 221.431,Z 699.145,A -85,B 0,C 180,E1 -20808.026,E2 -20808.026} C_VEL
LIN {X 0,Y 222.337,Z 707.125,A -85,B 0,C 180,E1 -20809.383,E2 -20809.383} C_VEL
LIN {X 0,Y 220.453,Z 717.576,A -85,B 0,C 180,E1 -20811.237,E2 -20811.237} C_VEL
LIN {X 0,Y 218.408,Z 727.689,A -85,B 0,C 180,E1 -20813.465,E2 -20813.465} C_VEL
LIN {X 0,Y 216.405,Z 736.875,A -85,B 0,C 180,E1 -20816.015,E2 -20816.015} C_VEL
LIN {X 0,Y 214.723,Z 744.642,A -85,B 0,C 180,E1 -20818.706,E2 -20818.706} C_VEL
LIN {X 0,Y 213.563,Z 750.381,A -85,B 0,C 180,E1 -20821.172,E2 -20821.172} C_VEL
LIN {X 0,Y 212.472,Z 756.037,A -85,B 0,C 180,E1 -20824.215,E2 -20824.215} C_VEL
LIN {X 0,Y 211.694,Z 760.2,A -85,B 0,C 180,E1 -20827.177,E2 -20827.177} C_VEL
LIN {X 0,Y 211.192,Z 763.157,A -85,B 0,C 180,E1 -20830.058,E2 -20830.058} C_VEL
LIN {X 0,Y 211.023,Z 765.1,A -85,B 0,C 180,E1 -20832.887,E2 -20832.887} C_VEL
LIN {X 0,Y 211.062,Z 766.109,A -85,B 0,C 180,E1 -20835.632,E2 -20835.632} C_VEL
LIN {X 0,Y 211.359,Z 766.296,A -85,B 0,C 180,E1 -20838.315,E2 -20838.315} C_VEL
LIN {X 0,Y 211.891,Z 765.737,A -85,B 0,C 180,E1 -20840.935,E2 -20840.935} C_VEL
LIN {X 0,Y 212.706,Z 764.469,A -85,B 0,C 180,E1 -20843.506,E2 -20843.506} C_VEL
LIN {X 0,Y 214.41,Z 761.25,A -85,B 0,C 180,E1 -20847.194,E2 -20847.194} C_VEL
LIN {X 0,Y 216.801,Z 756.253,A -85,B 0,C 180,E1 -20850.905,E2 -20850.905} C_VEL
LIN {X 0,Y 219.322,Z 750.848,A -85,B 0,C 180,E1 -20853.795,E2 -20853.795} C_VEL
LIN {X 0,Y 222.223,Z 744.311,A -85,B 0,C 180,E1 -20856.511,E2 -20856.511} C_VEL
LIN {X 0,Y 225.585,Z 736.159,A -85,B 0,C 180,E1 -20859.166,E2 -20859.166} C_VEL
LIN {X 0,Y 228.997,Z 727.123,A -85,B 0,C 180,E1 -20861.46,E2 -20861.46} C_VEL
LIN {X 0,Y 231.987,Z 718.246,A -85,B 0,C 180,E1 -20863.274,E2 -20863.274} C_VEL
LIN {X 0,Y 232.004,Z 710.559,A -85,B 0,C 180,E1 -20865.079,E2 -20865.079} C_VEL
LIN {X 0,Y 231.028,Z 700.966,A -85,B 0,C 180,E1 -20867.258,E2 -20867.258} C_VEL
LIN {X 0,Y 228.607,Z 689.722,A -85,B 0,C 180,E1 -20869.818,E2 -20869.818} C_VEL
LIN {X 0,Y 225.972,Z 681.759,A -85,B 0,C 180,E1 -20871.73,E2 -20871.73} C_VEL
LIN {X 0,Y 223.487,Z 676.161,A -85,B 0,C 180,E1 -20873.227,E2 -20873.227} C_VEL
LIN {X 0,Y 221.119,Z 671.836,A -85,B 0,C 180,E1 -20874.528,E2 -20874.528} C_VEL
LIN {X 0,Y 219.059,Z 668.471,A -85,B 0,C 180,E1 -20875.631,E2 -20875.631} C_VEL
LIN {X 0,Y 218.24,Z 667.02,A -85,B 0,C 180,E1 -20876.09,E2 -20876.09} C_VEL
LIN {X 0,Y 216.099,Z 664.121,A -85,B 0,C 180,E1 -20877.204,E2 -20877.204} C_VEL
LIN {X 0,Y 215.257,Z 661.885,A -85,B 0,C 180,E1 -20877.778,E2 -20877.778} C_VEL
LIN {X 0,Y 215.144,Z 660.444,A -85,B 0,C 180,E1 -20880,E2 -20880} C_VEL
LIN {X 0,Y 214.783,Z 659.317,A -85,B 0,C 180,E1 -20881.875,E2 -20881.875} C_VEL
LIN {X 0,Y 214.12,Z 657.813,A -85,B 0,C 180,E1 -20885.179,E2 -20885.179} C_VEL
LIN {X 0,Y 214.232,Z 657.797,A -85,B 0,C 180,E1 -20887.54,E2 -20887.54} C_VEL
LIN {X 0,Y 214.045,Z 657.821,A -85,B 0,C 180,E1 -20891.362,E2 -20891.362} C_VEL
LIN {X 0,Y 213.931,Z 657.838,A -85,B 0,C 180,E1 -20895.237,E2 -20895.237} C_VEL
LIN {X 0,Y 213.837,Z 657.845,A -85,B 0,C 180,E1 -20899.188,E2 -20899.188} C_VEL
LIN {X 0,Y 213.845,Z 657.845,A -85,B 0,C 180,E1 -20903.227,E2 -20903.227} C_VEL
LIN {X 0,Y 213.826,Z 657.851,A -85,B 0,C 180,E1 -20907.45,E2 -20907.45} C_VEL
LIN {X 0,Y 213.775,Z 657.856,A -85,B 0,C 180,E1 -20911.736,E2 -20911.736} C_VEL
LIN {X 0,Y 213.742,Z 657.859,A -85,B 0,C 180,E1 -20916.289,E2 -20916.289} C_VEL
LIN {X 0,Y 213.75,Z 658.02,A -85,B 0,C 180,E1 -20918.96,E2 -20918.96} C_VEL
LIN {X 0,Y 214.583,Z 660.48,A -85,B 0,C 180,E1 -20922.176,E2 -20922.176} C_VEL
LIN {X 0,Y 215.485,Z 664.981,A -85,B 0,C 180,E1 -20926.374,E2 -20926.374} C_VEL
LIN {X 0,Y 218.101,Z 669.345,A -85,B 0,C 180,E1 -20927.755,E2 -20927.755} C_VEL
LIN {X 0,Y 219.483,Z 671.304,A -85,B 0,C 180,E1 -20928.433,E2 -20928.433} C_VEL
LIN {X 0,Y 222.026,Z 676.079,A -85,B 0,C 180,E1 -20929.764,E2 -20929.764} C_VEL
LIN {X 0,Y 224.031,Z 680.754,A -85,B 0,C 180,E1 -20930.877,E2 -20930.877} C_VEL
LIN {X 0,Y 225.374,Z 684.864,A -85,B 0,C 180,E1 -20931.747,E2 -20931.747} C_VEL
LIN {X 0,Y 226.128,Z 687.928,A -85,B 0,C 180,E1 -20932.337,E2 -20932.337} C_VEL
LIN {X 0,Y 226.312,Z 693.057,A -85,B 0,C 180,E1 -20933.083,E2 -20933.083} C_VEL
LIN {X 0,Y 224.551,Z 705.639,A -85,B 0,C 180,E1 -20934.628,E2 -20934.628} C_VEL
LIN {X 0,Y 223.98,Z 710.731,A -85,B 0,C 180,E1 -20935.445,E2 -20935.445} C_VEL
LIN {X 0,Y 223.965,Z 712.31,A -85,B 0,C 180,E1 -20935.764,E2 -20935.764} C_VEL
LIN {X 0,Y 223.874,Z 722.363,A -85,B 0,C 180,E1 -20937.952,E2 -20937.952} C_VEL
LIN {X 0,Y 223.085,Z 730.179,A -85,B 0,C 180,E1 -20939.732,E2 -20939.732} C_VEL
LIN {X 0,Y 222.006,Z 735.918,A -85,B 0,C 180,E1 -20941.135,E2 -20941.135} C_VEL
LIN {X 0,Y 218.137,Z 746.018,A -85,B 0,C 180,E1 -20943.705,E2 -20943.705} C_VEL
LIN {X 0,Y 214.589,Z 754.153,A -85,B 0,C 180,E1 -20946.348,E2 -20946.348} C_VEL
LIN {X 0,Y 212.113,Z 759.781,A -85,B 0,C 180,E1 -20948.626,E2 -20948.626} C_VEL
LIN {X 0,Y 209.676,Z 765.309,A -85,B 0,C 180,E1 -20951.433,E2 -20951.433} C_VEL
LIN {X 0,Y 207.498,Z 769.698,A -85,B 0,C 180,E1 -20954.279,E2 -20954.279} C_VEL
LIN {X 0,Y 205.701,Z 773.962,A -85,B 0,C 180,E1 -20958.172,E2 -20958.172} C_VEL
LIN {X 0,Y 205.09,Z 775.456,A -85,B 0,C 180,E1 -20960.135,E2 -20960.135} C_VEL
LIN {X 0,Y 204.415,Z 777.221,A -85,B 0,C 180,E1 -20964.081,E2 -20964.081} C_VEL
LIN {X 0,Y 204.345,Z 777.53,A -85,B 0,C 180,E1 -20966.057,E2 -20966.057} C_VEL
LIN {X 0,Y 204.416,Z 777.422,A -85,B 0,C 180,E1 -20968.031,E2 -20968.031} C_VEL
LIN {X 0,Y 204.5,Z 778.259,A -85,B 0,C 180,E1 -20970.001,E2 -20970.001} C_VEL
LIN {X 0,Y 204.362,Z 778.792,A -85,B 0,C 180,E1 -20971.972,E2 -20971.972} C_VEL
LIN {X 0,Y 204.322,Z 778.918,A -85,B 0,C 180,E1 -20974.045,E2 -20974.045} C_VEL
LIN {X 0,Y 204.672,Z 777.965,A -85,B 0,C 180,E1 -20977.895,E2 -20977.895} C_VEL
LIN {X 0,Y 205.722,Z 775.473,A -85,B 0,C 180,E1 -20981.829,E2 -20981.829} C_VEL
LIN {X 0,Y 207.537,Z 771.285,A -85,B 0,C 180,E1 -20985.719,E2 -20985.719} C_VEL
LIN {X 0,Y 209.727,Z 766.993,A -85,B 0,C 180,E1 -20988.564,E2 -20988.564} C_VEL
LIN {X 0,Y 212.295,Z 761.585,A -85,B 0,C 180,E1 -20991.356,E2 -20991.356} C_VEL
LIN {X 0,Y 215.097,Z 755.153,A -85,B 0,C 180,E1 -20994.004,E2 -20994.004} C_VEL
LIN {X 0,Y 218.782,Z 746.711,A -85,B 0,C 180,E1 -20996.727,E2 -20996.727} C_VEL
LIN {X 0,Y 222.834,Z 736.578,A -85,B 0,C 180,E1 -20999.266,E2 -20999.266} C_VEL
LIN {X 0,Y 224.003,Z 728.815,A -85,B 0,C 180,E1 -21001.184,E2 -21001.184} C_VEL
LIN {X 0,Y 224.401,Z 720.518,A -85,B 0,C 180,E1 -21003.128,E2 -21003.128} C_VEL
LIN {X 0,Y 223.903,Z 711.04,A -85,B 0,C 180,E1 -21005.303,E2 -21005.303} C_VEL
LIN {X 0,Y 222.461,Z 701.668,A -85,B 0,C 180,E1 -21007.462,E2 -21007.462} C_VEL
LIN {X 0,Y 220.085,Z 692.742,A -85,B 0,C 180,E1 -21009.693,E2 -21009.693} C_VEL
LIN {X 0,Y 217.745,Z 686.87,A -85,B 0,C 180,E1 -21011.373,E2 -21011.373} C_VEL
LIN {X 0,Y 215.833,Z 682.907,A -85,B 0,C 180,E1 -21012.666,E2 -21012.666} C_VEL
LIN {X 0,Y 213.111,Z 678.155,A -85,B 0,C 180,E1 -21014.424,E2 -21014.424} C_VEL
LIN {X 0,Y 212.346,Z 676.405,A -85,B 0,C 180,E1 -21014.967,E2 -21014.967} C_VEL
LIN {X 0,Y 209.762,Z 673.122,A -85,B 0,C 180,E1 -21016.619,E2 -21016.619} C_VEL
LIN {X 0,Y 208.666,Z 670.222,A -85,B 0,C 180,E1 -21017.572,E2 -21017.572} C_VEL
LIN {X 0,Y 208.416,Z 668.604,A -85,B 0,C 180,E1 -21020.859,E2 -21020.859} C_VEL
LIN {X 0,Y 208.177,Z 666.882,A -85,B 0,C 180,E1 -21024.976,E2 -21024.976} C_VEL
LIN {X 0,Y 207.912,Z 665.389,A -85,B 0,C 180,E1 -21029.533,E2 -21029.533} C_VEL
LIN {X 0,Y 207.8,Z 664.352,A -85,B 0,C 180,E1 -21033.917,E2 -21033.917} C_VEL
LIN {X 0,Y 207.719,Z 663.741,A -85,B 0,C 180,E1 -21038.15,E2 -21038.15} C_VEL
LIN {X 0,Y 207.776,Z 663.494,A -85,B 0,C 180,E1 -21042.276,E2 -21042.276} C_VEL
LIN {X 0,Y 207.822,Z 663.605,A -85,B 0,C 180,E1 -21046.307,E2 -21046.307} C_VEL
LIN {X 0,Y 208.048,Z 663.985,A -85,B 0,C 180,E1 -21050.276,E2 -21050.276} C_VEL
LIN {X 0,Y 208.187,Z 664.692,A -85,B 0,C 180,E1 -21054.188,E2 -21054.188} C_VEL
LIN {X 0,Y 208.518,Z 665.626,A -85,B 0,C 180,E1 -21057.525,E2 -21057.525} C_VEL
LIN {X 0,Y 209.817,Z 668.411,A -85,B 0,C 180,E1 -21058.56,E2 -21058.56} C_VEL
LIN {X 0,Y 212.464,Z 671.286,A -85,B 0,C 180,E1 -21060.237,E2 -21060.237} C_VEL
LIN {X 0,Y 214.164,Z 674.736,A -85,B 0,C 180,E1 -21061.469,E2 -21061.469} C_VEL
LIN {X 0,Y 215.522,Z 676.67,A -85,B 0,C 180,E1 -21062.302,E2 -21062.302} C_VEL
LIN {X 0,Y 220.172,Z 685.973,A -85,B 0,C 180,E1 -21065.495,E2 -21065.495} C_VEL
LIN {X 0,Y 222.744,Z 693.411,A -85,B 0,C 180,E1 -21067.639,E2 -21067.639} C_VEL
LIN {X 0,Y 224.897,Z 702.046,A -85,B 0,C 180,E1 -21069.933,E2 -21069.933} C_VEL
LIN {X 0,Y 226.207,Z 712.222,A -85,B 0,C 180,E1 -21072.561,E2 -21072.561} C_VEL
LIN {X 0,Y 226.247,Z 721.091,A -85,B 0,C 180,E1 -21074.849,E2 -21074.849} C_VEL
LIN {X 0,Y 222.549,Z 731.124,A -85,B 0,C 180,E1 -21077.107,E2 -21077.107} C_VEL
LIN {X 0,Y 218.874,Z 739.76,A -85,B 0,C 180,E1 -21079.538,E2 -21079.538} C_VEL
LIN {X 0,Y 215.649,Z 746.753,A -85,B 0,C 180,E1 -21082.011,E2 -21082.011} C_VEL
LIN {X 0,Y 212.508,Z 753.19,A -85,B 0,C 180,E1 -21084.939,E2 -21084.939} C_VEL
LIN {X 0,Y 209.89,Z 758.263,A -85,B 0,C 180,E1 -21087.955,E2 -21087.955} C_VEL
LIN {X 0,Y 208.135,Z 761.474,A -85,B 0,C 180,E1 -21090.431,E2 -21090.431} C_VEL
LIN {X 0,Y 206.772,Z 763.91,A -85,B 0,C 180,E1 -21092.945,E2 -21092.945} C_VEL
LIN {X 0,Y 205.692,Z 765.669,A -85,B 0,C 180,E1 -21095.511,E2 -21095.511} C_VEL
LIN {X 0,Y 204.886,Z 766.778,A -85,B 0,C 180,E1 -21098.129,E2 -21098.129} C_VEL
LIN {X 0,Y 204.356,Z 767.154,A -85,B 0,C 180,E1 -21100.834,E2 -21100.834} C_VEL
LIN {X 0,Y 204.052,Z 766.758,A -85,B 0,C 180,E1 -21103.673,E2 -21103.673} C_VEL
LIN {X 0,Y 204.035,Z 765.588,A -85,B 0,C 180,E1 -21106.456,E2 -21106.456} C_VEL
LIN {X 0,Y 204.298,Z 763.668,A -85,B 0,C 180,E1 -21109.185,E2 -21109.185} C_VEL
LIN {X 0,Y 204.75,Z 760.644,A -85,B 0,C 180,E1 -21112.136,E2 -21112.136} C_VEL
LIN {X 0,Y 205.532,Z 756.453,A -85,B 0,C 180,E1 -21115.151,E2 -21115.151} C_VEL
LIN {X 0,Y 206.61,Z 750.806,A -85,B 0,C 180,E1 -21118.255,E2 -21118.255} C_VEL
LIN {X 0,Y 208.176,Z 743.53,A -85,B 0,C 180,E1 -21121.373,E2 -21121.373} C_VEL
LIN {X 0,Y 210.065,Z 735.135,A -85,B 0,C 180,E1 -21124.218,E2 -21124.218} C_VEL
LIN {X 0,Y 212.268,Z 725.309,A -85,B 0,C 180,E1 -21126.838,E2 -21126.838} C_VEL
LIN {X 0,Y 214.54,Z 714.514,A -85,B 0,C 180,E1 -21129.129,E2 -21129.129} C_VEL
LIN {X 0,Y 215.551,Z 708.32,A -85,B 0,C 180,E1 -21130.227,E2 -21130.227} C_VEL
LIN {X 0,Y 214.185,Z 697.503,A -85,B 0,C 180,E1 -21132.135,E2 -21132.135} C_VEL
LIN {X 0,Y 212.093,Z 685.846,A -85,B 0,C 180,E1 -21133.886,E2 -21133.886} C_VEL
LIN {X 0,Y 209.197,Z 673.287,A -85,B 0,C 180,E1 -21135.468,E2 -21135.468} C_VEL
LIN {X 0,Y 206.269,Z 662.229,A -85,B 0,C 180,E1 -21136.64,E2 -21136.64} C_VEL
LIN {X 0,Y 207.1,Z 658.686,A -85,B 0,C 180,E1 -21141.499,E2 -21141.499} C_VEL
LIN {X 0,Y 207.385,Z 658.648,A -85,B 0,C 180,E1 -21148.057,E2 -21148.057} C_VEL
LIN {X 0,Y 207.518,Z 658.635,A -85,B 0,C 180,E1 -21149.999,E2 -21149.999} C_VEL
LIN {X 0,Y 207.382,Z 658.647,A -85,B 0,C 180,E1 -21151.941,E2 -21151.941} C_VEL
LIN {X 0,Y 206.984,Z 658.695,A -85,B 0,C 180,E1 -21157.805,E2 -21157.805} C_VEL
LIN {X 0,Y 206.576,Z 658.764,A -85,B 0,C 180,E1 -21161.032,E2 -21161.032} C_VEL
LIN {X 0,Y 206.282,Z 660.26,A -85,B 0,C 180,E1 -21162.481,E2 -21162.481} C_VEL
LIN {X 0,Y 209.996,Z 675.031,A -85,B 0,C 180,E1 -21163.992,E2 -21163.992} C_VEL
LIN {X 0,Y 212.591,Z 687.503,A -85,B 0,C 180,E1 -21165.58,E2 -21165.58} C_VEL
LIN {X 0,Y 214.483,Z 699.541,A -85,B 0,C 180,E1 -21167.421,E2 -21167.421} C_VEL
LIN {X 0,Y 215.473,Z 708.017,A -85,B 0,C 180,E1 -21168.935,E2 -21168.935} C_VEL
LIN {X 0,Y 213.399,Z 719.052,A -85,B 0,C 180,E1 -21170.986,E2 -21170.986} C_VEL
LIN {X 0,Y 211.421,Z 728.355,A -85,B 0,C 180,E1 -21173.144,E2 -21173.144} C_VEL
LIN {X 0,Y 209.274,Z 737.8,A -85,B 0,C 180,E1 -21175.885,E2 -21175.885} C_VEL
LIN {X 0,Y 207.478,Z 745.92,A -85,B 0,C 180,E1 -21178.861,E2 -21178.861} C_VEL
LIN {X 0,Y 206.255,Z 751.801,A -85,B 0,C 180,E1 -21181.585,E2 -21181.585} C_VEL
LIN {X 0,Y 205.196,Z 757.106,A -85,B 0,C 180,E1 -21184.714,E2 -21184.714} C_VEL
LIN {X 0,Y 204.381,Z 761.543,A -85,B 0,C 180,E1 -21188.239,E2 -21188.239} C_VEL
LIN {X 0,Y 203.999,Z 763.888,A -85,B 0,C 180,E1 -21190.886,E2 -21190.886} C_VEL
LIN {X 0,Y 203.932,Z 765.532,A -85,B 0,C 180,E1 -21193.638,E2 -21193.638} C_VEL
LIN {X 0,Y 204.031,Z 766.412,A -85,B 0,C 180,E1 -21196.455,E2 -21196.455} C_VEL
LIN {X 0,Y 204.428,Z 766.479,A -85,B 0,C 180,E1 -21199.217,E2 -21199.217} C_VEL
LIN {X 0,Y 205.106,Z 765.736,A -85,B 0,C 180,E1 -21202.006,E2 -21202.006} C_VEL
LIN {X 0,Y 206.161,Z 764.121,A -85,B 0,C 180,E1 -21204.899,E2 -21204.899} C_VEL
LIN {X 0,Y 207.624,Z 761.577,A -85,B 0,C 180,E1 -21207.803,E2 -21207.803} C_VEL
LIN {X 0,Y 210.034,Z 756.964,A -85,B 0,C 180,E1 -21211.441,E2 -21211.441} C_VEL
LIN {X 0,Y 212.835,Z 751.362,A -85,B 0,C 180,E1 -21214.578,E2 -21214.578} C_VEL
LIN {X 0,Y 216.094,Z 744.441,A -85,B 0,C 180,E1 -21217.534,E2 -21217.534} C_VEL
LIN {X 0,Y 219.103,Z 737.625,A -85,B 0,C 180,E1 -21219.829,E2 -21219.829} C_VEL
LIN {X 0,Y 222.69,Z 728.914,A -85,B 0,C 180,E1 -21222.188,E2 -21222.188} C_VEL
LIN {X 0,Y 225.955,Z 719.798,A -85,B 0,C 180,E1 -21224.161,E2 -21224.161} C_VEL
LIN {X 0,Y 226.08,Z 712.205,A -85,B 0,C 180,E1 -21226.059,E2 -21226.059} C_VEL
LIN {X 0,Y 225.333,Z 703.205,A -85,B 0,C 180,E1 -21228.24,E2 -21228.24} C_VEL
LIN {X 0,Y 223.587,Z 693.979,A -85,B 0,C 180,E1 -21230.501,E2 -21230.501} C_VEL
LIN {X 0,Y 221.071,Z 685.455,A -85,B 0,C 180,E1 -21232.694,E2 -21232.694} C_VEL
LIN {X 0,Y 217.51,Z 677.576,A -85,B 0,C 180,E1 -21235.077,E2 -21235.077} C_VEL
LIN {X 0,Y 215.418,Z 673.875,A -85,B 0,C 180,E1 -21236.376,E2 -21236.376} C_VEL
LIN {X 0,Y 214.364,Z 672.203,A -85,B 0,C 180,E1 -21237.005,E2 -21237.005} C_VEL
LIN {X 0,Y 212.245,Z 668.439,A -85,B 0,C 180,E1 -21238.363,E2 -21238.363} C_VEL
LIN {X 0,Y 211.608,Z 667.438,A -85,B 0,C 180,E1 -21238.763,E2 -21238.763} C_VEL
LIN {X 0,Y 209.116,Z 664.137,A -85,B 0,C 180,E1 -21240.301,E2 -21240.301} C_VEL
LIN {X 0,Y 208.254,Z 662.195,A -85,B 0,C 180,E1 -21240.967,E2 -21240.967} C_VEL
LIN {X 0,Y 207.145,Z 658.682,A -85,B 0,C 180,E1 -21248.291,E2 -21248.291} C_VEL
LIN {X 0,Y 206.98,Z 658.7,A -85,B 0,C 180,E1 -21251.755,E2 -21251.755} C_VEL
LIN {X 0,Y 206.864,Z 658.716,A -85,B 0,C 180,E1 -21255.771,E2 -21255.771} C_VEL
LIN {X 0,Y 206.781,Z 658.727,A -85,B 0,C 180,E1 -21259.869,E2 -21259.869} C_VEL
LIN {X 0,Y 206.761,Z 658.726,A -85,B 0,C 180,E1 -21264.072,E2 -21264.072} C_VEL
LIN {X 0,Y 206.741,Z 658.729,A -85,B 0,C 180,E1 -21268.419,E2 -21268.419} C_VEL
LIN {X 0,Y 206.701,Z 658.734,A -85,B 0,C 180,E1 -21272.957,E2 -21272.957} C_VEL
LIN {X 0,Y 206.734,Z 658.958,A -85,B 0,C 180,E1 -21275.142,E2 -21275.142} C_VEL
LIN {X 0,Y 207.621,Z 662.045,A -85,B 0,C 180,E1 -21280.027,E2 -21280.027} C_VEL
LIN {X 0,Y 208.419,Z 664.64,A -85,B 0,C 180,E1 -21283.107,E2 -21283.107} C_VEL
LIN {X 0,Y 211.05,Z 669.191,A -85,B 0,C 180,E1 -21284.852,E2 -21284.852} C_VEL
LIN {X 0,Y 212.676,Z 671.359,A -85,B 0,C 180,E1 -21285.782,E2 -21285.782} C_VEL
LIN {X 0,Y 215.374,Z 675.816,A -85,B 0,C 180,E1 -21287.358,E2 -21287.358} C_VEL
LIN {X 0,Y 218.122,Z 681.28,A -85,B 0,C 180,E1 -21288.996,E2 -21288.996} C_VEL
LIN {X 0,Y 219.775,Z 685.725,A -85,B 0,C 180,E1 -21290.128,E2 -21290.128} C_VEL
LIN {X 0,Y 221.678,Z 693.419,A -85,B 0,C 180,E1 -21291.809,E2 -21291.809} C_VEL
LIN {X 0,Y 223.396,Z 704.282,A -85,B 0,C 180,E1 -21294.092,E2 -21294.092} C_VEL
LIN {X 0,Y 223.965,Z 712.31,A -85,B 0,C 180,E1 -21295.764,E2 -21295.764} C_VEL
LIN {X 0,Y 223.539,Z 717.117,A -85,B 0,C 180,E1 -21296.676,E2 -21296.676} C_VEL
LIN {X 0,Y 222.207,Z 721.999,A -85,B 0,C 180,E1 -21297.487,E2 -21297.487} C_VEL
LIN {X 0,Y 218.223,Z 731.498,A -85,B 0,C 180,E1 -21299.079,E2 -21299.079} C_VEL
LIN {X 0,Y 215.728,Z 737.389,A -85,B 0,C 180,E1 -21300.336,E2 -21300.336} C_VEL
LIN {X 0,Y 211.854,Z 746.791,A -85,B 0,C 180,E1 -21302.863,E2 -21302.863} C_VEL
LIN {X 0,Y 208.136,Z 754.736,A -85,B 0,C 180,E1 -21305.567,E2 -21305.567} C_VEL
LIN {X 0,Y 205.523,Z 760.2,A -85,B 0,C 180,E1 -21307.905,E2 -21307.905} C_VEL
LIN {X 0,Y 202.955,Z 765.595,A -85,B 0,C 180,E1 -21310.795,E2 -21310.795} C_VEL
LIN {X 0,Y 200.666,Z 769.873,A -85,B 0,C 180,E1 -21313.73,E2 -21313.73} C_VEL
LIN {X 0,Y 199.568,Z 772.154,A -85,B 0,C 180,E1 -21315.73,E2 -21315.73} C_VEL
LIN {X 0,Y 198.719,Z 774.006,A -85,B 0,C 180,E1 -21317.75,E2 -21317.75} C_VEL
LIN {X 0,Y 197.599,Z 776.44,A -85,B 0,C 180,E1 -21321.822,E2 -21321.822} C_VEL
LIN {X 0,Y 197.35,Z 777.087,A -85,B 0,C 180,E1 -21323.868,E2 -21323.868} C_VEL
LIN {X 0,Y 197.286,Z 777.333,A -85,B 0,C 180,E1 -21325.915,E2 -21325.915} C_VEL
LIN {X 0,Y 197.317,Z 777.157,A -85,B 0,C 180,E1 -21327.96,E2 -21327.96} C_VEL
LIN {X 0,Y 197.417,Z 777.929,A -85,B 0,C 180,E1 -21330.001,E2 -21330.001} C_VEL
LIN {X 0,Y 197.248,Z 778.693,A -85,B 0,C 180,E1 -21333.928,E2 -21333.928} C_VEL
LIN {X 0,Y 197.367,Z 778.489,A -85,B 0,C 180,E1 -21336.133,E2 -21336.133} C_VEL
LIN {X 0,Y 198.075,Z 776.861,A -85,B 0,C 180,E1 -21340.22,E2 -21340.22} C_VEL
LIN {X 0,Y 199.612,Z 773.699,A -85,B 0,C 180,E1 -21344.269,E2 -21344.269} C_VEL
LIN {X 0,Y 201.426,Z 770.199,A -85,B 0,C 180,E1 -21347.253,E2 -21347.253} C_VEL
LIN {X 0,Y 203.932,Z 765.659,A -85,B 0,C 180,E1 -21350.16,E2 -21350.16} C_VEL
LIN {X 0,Y 206.774,Z 759.602,A -85,B 0,C 180,E1 -21353.209,E2 -21353.209} C_VEL
LIN {X 0,Y 210.545,Z 751.711,A -85,B 0,C 180,E1 -21356.251,E2 -21356.251} C_VEL
LIN {X 0,Y 214.604,Z 742.871,A -85,B 0,C 180,E1 -21358.885,E2 -21358.885} C_VEL
LIN {X 0,Y 216.721,Z 737.683,A -85,B 0,C 180,E1 -21360.176,E2 -21360.176} C_VEL
LIN {X 0,Y 217.996,Z 730.133,A -85,B 0,C 180,E1 -21362.147,E2 -21362.147} C_VEL
LIN {X 0,Y 218.557,Z 722.075,A -85,B 0,C 180,E1 -21364.161,E2 -21364.161} C_VEL
LIN {X 0,Y 218.234,Z 713.06,A -85,B 0,C 180,E1 -21366.38,E2 -21366.38} C_VEL
LIN {X 0,Y 217.016,Z 703.783,A -85,B 0,C 180,E1 -21368.706,E2 -21368.706} C_VEL
LIN {X 0,Y 215.077,Z 696.092,A -85,B 0,C 180,E1 -21370.809,E2 -21370.809} C_VEL
LIN {X 0,Y 212.144,Z 688.845,A -85,B 0,C 180,E1 -21373.212,E2 -21373.212} C_VEL
LIN {X 0,Y 209.219,Z 682.676,A -85,B 0,C 180,E1 -21375.489,E2 -21375.489} C_VEL
LIN {X 0,Y 206.491,Z 678.53,A -85,B 0,C 180,E1 -21377.51,E2 -21377.51} C_VEL
LIN {X 0,Y 205.515,Z 676.263,A -85,B 0,C 180,E1 -21378.379,E2 -21378.379} C_VEL
LIN {X 0,Y 202.911,Z 673.272,A -85,B 0,C 180,E1 -21380.437,E2 -21380.437} C_VEL
LIN {X 0,Y 201.477,Z 670.074,A -85,B 0,C 180,E1 -21381.905,E2 -21381.905} C_VEL
LIN {X 0,Y 201.403,Z 669.669,A -85,B 0,C 180,E1 -21382.047,E2 -21382.047} C_VEL
LIN {X 0,Y 201.123,Z 667.822,A -85,B 0,C 180,E1 -21386.999,E2 -21386.999} C_VEL
LIN {X 0,Y 200.973,Z 666.696,A -85,B 0,C 180,E1 -21390.957,E2 -21390.957} C_VEL
LIN {X 0,Y 200.879,Z 665.81,A -85,B 0,C 180,E1 -21395.457,E2 -21395.457} C_VEL
LIN {X 0,Y 200.787,Z 665.359,A -85,B 0,C 180,E1 -21399.511,E2 -21399.511} C_VEL
LIN {X 0,Y 200.891,Z 665.213,A -85,B 0,C 180,E1 -21403.747,E2 -21403.747} C_VEL
LIN {X 0,Y 201.02,Z 665.45,A -85,B 0,C 180,E1 -21408.219,E2 -21408.219} C_VEL
LIN {X 0,Y 201.252,Z 666.183,A -85,B 0,C 180,E1 -21412.98,E2 -21412.98} C_VEL
LIN {X 0,Y 202.361,Z 668.716,A -85,B 0,C 180,E1 -21414.207,E2 -21414.207} C_VEL
LIN {X 0,Y 204.75,Z 671.287,A -85,B 0,C 180,E1 -21416.187,E2 -21416.187} C_VEL
LIN {X 0,Y 205.772,Z 672.162,A -85,B 0,C 180,E1 -21416.941,E2 -21416.941} C_VEL
LIN {X 0,Y 207.621,Z 675.515,A -85,B 0,C 180,E1 -21418.51,E2 -21418.51} C_VEL
LIN {X 0,Y 209.059,Z 676.946,A -85,B 0,C 180,E1 -21419.47,E2 -21419.47} C_VEL
LIN {X 0,Y 210.874,Z 680.8,A -85,B 0,C 180,E1 -21421.009,E2 -21421.009} C_VEL
LIN {X 0,Y 212.087,Z 682.966,A -85,B 0,C 180,E1 -21421.899,E2 -21421.899} C_VEL
LIN {X 0,Y 215.159,Z 689.469,A -85,B 0,C 180,E1 -21424.349,E2 -21424.349} C_VEL
LIN {X 0,Y 217.391,Z 695.997,A -85,B 0,C 180,E1 -21426.419,E2 -21426.419} C_VEL
LIN {X 0,Y 219.476,Z 705.696,A -85,B 0,C 180,E1 -21429.213,E2 -21429.213} C_VEL
LIN {X 0,Y 220.333,Z 713.976,A -85,B 0,C 180,E1 -21431.5,E2 -21431.5} C_VEL
LIN {X 0,Y 220.28,Z 722.362,A -85,B 0,C 180,E1 -21433.833,E2 -21433.833} C_VEL
LIN {X 0,Y 219.128,Z 725.878,A -85,B 0,C 180,E1 -21434.627,E2 -21434.627} C_VEL
LIN {X 0,Y 215,Z 735.699,A -85,B 0,C 180,E1 -21437.109,E2 -21437.109} C_VEL
LIN {X 0,Y 211.596,Z 742.904,A -85,B 0,C 180,E1 -21439.399,E2 -21439.399} C_VEL
LIN {X 0,Y 208.625,Z 748.847,A -85,B 0,C 180,E1 -21441.75,E2 -21441.75} C_VEL
LIN {X 0,Y 206.004,Z 753.795,A -85,B 0,C 180,E1 -21444.167,E2 -21444.167} C_VEL
LIN {X 0,Y 203.703,Z 757.922,A -85,B 0,C 180,E1 -21446.649,E2 -21446.649} C_VEL
LIN {X 0,Y 200.951,Z 762.611,A -85,B 0,C 180,E1 -21450.492,E2 -21450.492} C_VEL
LIN {X 0,Y 199.892,Z 764.354,A -85,B 0,C 180,E1 -21452.453,E2 -21452.453} C_VEL
LIN {X 0,Y 198.571,Z 766.234,A -85,B 0,C 180,E1 -21455.507,E2 -21455.507} C_VEL
LIN {X 0,Y 197.678,Z 767.201,A -85,B 0,C 180,E1 -21458.54,E2 -21458.54} C_VEL
LIN {X 0,Y 197.029,Z 767.154,A -85,B 0,C 180,E1 -21462.667,E2 -21462.667} C_VEL
LIN {X 0,Y 196.919,Z 766.168,A -85,B 0,C 180,E1 -21465.545,E2 -21465.545} C_VEL
LIN {X 0,Y 197.108,Z 764.314,A -85,B 0,C 180,E1 -21468.484,E2 -21468.484} C_VEL
LIN {X 0,Y 197.544,Z 761.499,A -85,B 0,C 180,E1 -21471.508,E2 -21471.508} C_VEL
LIN {X 0,Y 198.261,Z 757.545,A -85,B 0,C 180,E1 -21474.618,E2 -21474.618} C_VEL
LIN {X 0,Y 199.383,Z 751.734,A -85,B 0,C 180,E1 -21478.079,E2 -21478.079} C_VEL
LIN {X 0,Y 201.107,Z 743.999,A -85,B 0,C 180,E1 -21481.561,E2 -21481.561} C_VEL
LIN {X 0,Y 203.083,Z 735.509,A -85,B 0,C 180,E1 -21484.556,E2 -21484.556} C_VEL
LIN {X 0,Y 205.175,Z 726.543,A -85,B 0,C 180,E1 -21487.061,E2 -21487.061} C_VEL
LIN {X 0,Y 207.485,Z 715.984,A -85,B 0,C 180,E1 -21489.425,E2 -21489.425} C_VEL
LIN {X 0,Y 208.677,Z 709.929,A -85,B 0,C 180,E1 -21490.564,E2 -21490.564} C_VEL
LIN {X 0,Y 207.501,Z 699.449,A -85,B 0,C 180,E1 -21492.506,E2 -21492.506} C_VEL
LIN {X 0,Y 205.498,Z 687.702,A -85,B 0,C 180,E1 -21494.375,E2 -21494.375} C_VEL
LIN {X 0,Y 202.514,Z 674.377,A -85,B 0,C 180,E1 -21496.17,E2 -21496.17} C_VEL
LIN {X 0,Y 199.294,Z 662.429,A -85,B 0,C 180,E1 -21497.499,E2 -21497.499} C_VEL
LIN {X 0,Y 200.075,Z 659.561,A -85,B 0,C 180,E1 -21501.713,E2 -21501.713} C_VEL
LIN {X 0,Y 200.324,Z 659.528,A -85,B 0,C 180,E1 -21507.989,E2 -21507.989} C_VEL
LIN {X 0,Y 200.482,Z 659.511,A -85,B 0,C 180,E1 -21509.999,E2 -21509.999} C_VEL
LIN {X 0,Y 200.012,Z 659.567,A -85,B 0,C 180,E1 -21514.029,E2 -21514.029} C_VEL
LIN {X 0,Y 199.915,Z 659.576,A -85,B 0,C 180,E1 -21518.083,E2 -21518.083} C_VEL
LIN {X 0,Y 199.571,Z 659.683,A -85,B 0,C 180,E1 -21520.91,E2 -21520.91} C_VEL
LIN {X 0,Y 199.421,Z 660.428,A -85,B 0,C 180,E1 -21521.626,E2 -21521.626} C_VEL
LIN {X 0,Y 202.681,Z 673.424,A -85,B 0,C 180,E1 -21522.993,E2 -21522.993} C_VEL
LIN {X 0,Y 205.339,Z 685.826,A -85,B 0,C 180,E1 -21524.593,E2 -21524.593} C_VEL
LIN {X 0,Y 207.361,Z 698.064,A -85,B 0,C 180,E1 -21526.489,E2 -21526.489} C_VEL
LIN {X 0,Y 208.587,Z 709.251,A -85,B 0,C 180,E1 -21528.534,E2 -21528.534} C_VEL
LIN {X 0,Y 206.341,Z 720.295,A -85,B 0,C 180,E1 -21530.693,E2 -21530.693} C_VEL
LIN {X 0,Y 203.993,Z 730.888,A -85,B 0,C 180,E1 -21533.339,E2 -21533.339} C_VEL
LIN {X 0,Y 201.872,Z 739.807,A -85,B 0,C 180,E1 -21536.146,E2 -21536.146} C_VEL
LIN {X 0,Y 200.048,Z 748.015,A -85,B 0,C 180,E1 -21539.46,E2 -21539.46} C_VEL
LIN {X 0,Y 198.744,Z 754.154,A -85,B 0,C 180,E1 -21542.632,E2 -21542.632} C_VEL
LIN {X 0,Y 197.725,Z 759.307,A -85,B 0,C 180,E1 -21546.161,E2 -21546.161} C_VEL
LIN {X 0,Y 197.012,Z 763.247,A -85,B 0,C 180,E1 -21549.948,E2 -21549.948} C_VEL
LIN {X 0,Y 196.798,Z 765.151,A -85,B 0,C 180,E1 -21552.727,E2 -21552.727} C_VEL
LIN {X 0,Y 196.868,Z 766.328,A -85,B 0,C 180,E1 -21555.558,E2 -21555.558} C_VEL
LIN {X 0,Y 197.181,Z 766.752,A -85,B 0,C 180,E1 -21558.458,E2 -21558.458} C_VEL
LIN {X 0,Y 197.794,Z 766.359,A -85,B 0,C 180,E1 -21561.415,E2 -21561.415} C_VEL
LIN {X 0,Y 198.815,Z 765.097,A -85,B 0,C 180,E1 -21564.392,E2 -21564.392} C_VEL
LIN {X 0,Y 200.762,Z 762.066,A -85,B 0,C 180,E1 -21568.325,E2 -21568.325} C_VEL
LIN {X 0,Y 202.42,Z 759.158,A -85,B 0,C 180,E1 -21570.917,E2 -21570.917} C_VEL
LIN {X 0,Y 205.083,Z 754.329,A -85,B 0,C 180,E1 -21574.092,E2 -21574.092} C_VEL
LIN {X 0,Y 208.515,Z 747.783,A -85,B 0,C 180,E1 -21577.322,E2 -21577.322} C_VEL
LIN {X 0,Y 212.357,Z 739.83,A -85,B 0,C 180,E1 -21580.319,E2 -21580.319} C_VEL
LIN {X 0,Y 216.487,Z 730.47,A -85,B 0,C 180,E1 -21583.012,E2 -21583.012} C_VEL
LIN {X 0,Y 219.617,Z 722.552,A -85,B 0,C 180,E1 -21584.824,E2 -21584.824} C_VEL
LIN {X 0,Y 220.112,Z 719.205,A -85,B 0,C 180,E1 -21585.665,E2 -21585.665} C_VEL
LIN {X 0,Y 220.086,Z 710.625,A -85,B 0,C 180,E1 -21587.935,E2 -21587.935} C_VEL
LIN {X 0,Y 219.094,Z 701.529,A -85,B 0,C 180,E1 -21590.305,E2 -21590.305} C_VEL
LIN {X 0,Y 217.371,Z 693.079,A -85,B 0,C 180,E1 -21592.569,E2 -21592.569} C_VEL
LIN {X 0,Y 215.294,Z 686.994,A -85,B 0,C 180,E1 -21594.38,E2 -21594.38} C_VEL
LIN {X 0,Y 211.799,Z 679.688,A -85,B 0,C 180,E1 -21596.968,E2 -21596.968} C_VEL
LIN {X 0,Y 208.834,Z 673.897,A -85,B 0,C 180,E1 -21599.181,E2 -21599.181} C_VEL
LIN {X 0,Y 206.185,Z 670.026,A -85,B 0,C 180,E1 -21601.038,E2 -21601.038} C_VEL
LIN {X 0,Y 205.197,Z 668.233,A -85,B 0,C 180,E1 -21601.84,E2 -21601.84} C_VEL
LIN {X 0,Y 202.045,Z 665.167,A -85,B 0,C 180,E1 -21604.114,E2 -21604.114} C_VEL
LIN {X 0,Y 200.729,Z 662.511,A -85,B 0,C 180,E1 -21605.525,E2 -21605.525} C_VEL
LIN {X 0,Y 200.591,Z 661.396,A -85,B 0,C 180,E1 -21608.056,E2 -21608.056} C_VEL
LIN {X 0,Y 199.993,Z 660.147,A -85,B 0,C 180,E1 -21612.172,E2 -21612.172} C_VEL
LIN {X 0,Y 199.815,Z 659.596,A -85,B 0,C 180,E1 -21615.295,E2 -21615.295} C_VEL
LIN {X 0,Y 199.781,Z 659.597,A -85,B 0,C 180,E1 -21618.458,E2 -21618.458} C_VEL
LIN {X 0,Y 199.734,Z 659.601,A -85,B 0,C 180,E1 -21623.818,E2 -21623.818} C_VEL
LIN {X 0,Y 199.71,Z 659.623,A -85,B 0,C 180,E1 -21628.387,E2 -21628.387} C_VEL
LIN {X 0,Y 200.268,Z 661.709,A -85,B 0,C 180,E1 -21634.159,E2 -21634.159} C_VEL
LIN {X 0,Y 201.171,Z 664.625,A -85,B 0,C 180,E1 -21638.965,E2 -21638.965} C_VEL
LIN {X 0,Y 203.456,Z 668.353,A -85,B 0,C 180,E1 -21640.871,E2 -21640.871} C_VEL
LIN {X 0,Y 205.895,Z 671.2,A -85,B 0,C 180,E1 -21642.569,E2 -21642.569} C_VEL
LIN {X 0,Y 208.426,Z 675.594,A -85,B 0,C 180,E1 -21644.392,E2 -21644.392} C_VEL
LIN {X 0,Y 209.536,Z 677.313,A -85,B 0,C 180,E1 -21645.112,E2 -21645.112} C_VEL
LIN {X 0,Y 212.591,Z 683.003,A -85,B 0,C 180,E1 -21647.18,E2 -21647.18} C_VEL
LIN {X 0,Y 214.82,Z 688.399,A -85,B 0,C 180,E1 -21648.804,E2 -21648.804} C_VEL
LIN {X 0,Y 216.382,Z 694.771,A -85,B 0,C 180,E1 -21650.367,E2 -21650.367} C_VEL
LIN {X 0,Y 217.946,Z 705.906,A -85,B 0,C 180,E1 -21652.876,E2 -21652.876} C_VEL
LIN {X 0,Y 218.316,Z 715.93,A -85,B 0,C 180,E1 -21655.117,E2 -21655.117} C_VEL
LIN {X 0,Y 217.894,Z 725.069,A -85,B 0,C 180,E1 -21657.243,E2 -21657.243} C_VEL
LIN {X 0,Y 216.654,Z 733.322,A -85,B 0,C 180,E1 -21659.277,E2 -21659.277} C_VEL
LIN {X 0,Y 215.728,Z 737.389,A -85,B 0,C 180,E1 -21660.336,E2 -21660.336} C_VEL
LIN {X 0,Y 213.584,Z 741.61,A -85,B 0,C 180,E1 -21661.296,E2 -21661.296} C_VEL
LIN {X 0,Y 208.327,Z 748.15,A -85,B 0,C 180,E1 -21662.736,E2 -21662.736} C_VEL
LIN {X 0,Y 202.948,Z 754.114,A -85,B 0,C 180,E1 -21664.357,E2 -21664.357} C_VEL
LIN {X 0,Y 200.662,Z 757.357,A -85,B 0,C 180,E1 -21665.589,E2 -21665.589} C_VEL
LIN {X 0,Y 198.081,Z 762.542,A -85,B 0,C 180,E1 -21668.128,E2 -21668.128} C_VEL
LIN {X 0,Y 195.41,Z 767.411,A -85,B 0,C 180,E1 -21671.115,E2 -21671.115} C_VEL
LIN {X 0,Y 193.232,Z 771.204,A -85,B 0,C 180,E1 -21674.171,E2 -21674.171} C_VEL
LIN {X 0,Y 191.755,Z 774.027,A -85,B 0,C 180,E1 -21677.298,E2 -21677.298} C_VEL
LIN {X 0,Y 190.549,Z 776.361,A -85,B 0,C 180,E1 -21681.517,E2 -21681.517} C_VEL
LIN {X 0,Y 190.285,Z 776.948,A -85,B 0,C 180,E1 -21683.639,E2 -21683.639} C_VEL
LIN {X 0,Y 190.191,Z 777.092,A -85,B 0,C 180,E1 -21686.126,E2 -21686.126} C_VEL
LIN {X 0,Y 190.222,Z 776.88,A -85,B 0,C 180,E1 -21687.884,E2 -21687.884} C_VEL
LIN {X 0,Y 190.335,Z 777.599,A -85,B 0,C 180,E1 -21690.001,E2 -21690.001} C_VEL
LIN {X 0,Y 190.163,Z 778.46,A -85,B 0,C 180,E1 -21694.24,E2 -21694.24} C_VEL
LIN {X 0,Y 190.299,Z 778.318,A -85,B 0,C 180,E1 -21696.362,E2 -21696.362} C_VEL
LIN {X 0,Y 190.581,Z 777.773,A -85,B 0,C 180,E1 -21698.483,E2 -21698.483} C_VEL
LIN {X 0,Y 191.778,Z 775.493,A -85,B 0,C 180,E1 -21702.703,E2 -21702.703} C_VEL
LIN {X 0,Y 193.269,Z 772.74,A -85,B 0,C 180,E1 -21705.827,E2 -21705.827} C_VEL
LIN {X 0,Y 195.458,Z 769.027,A -85,B 0,C 180,E1 -21708.882,E2 -21708.882} C_VEL
LIN {X 0,Y 198.229,Z 764.274,A -85,B 0,C 180,E1 -21711.856,E2 -21711.856} C_VEL
LIN {X 0,Y 201.215,Z 758.372,A -85,B 0,C 180,E1 -21714.781,E2 -21714.781} C_VEL
LIN {X 0,Y 204.911,Z 751.097,A -85,B 0,C 180,E1 -21717.583,E2 -21717.583} C_VEL
LIN {X 0,Y 209.201,Z 742.183,A -85,B 0,C 180,E1 -21720.26,E2 -21720.26} C_VEL
LIN {X 0,Y 210.651,Z 738.777,A -85,B 0,C 180,E1 -21721.141,E2 -21721.141} C_VEL
LIN {X 0,Y 212.265,Z 730.246,A -85,B 0,C 180,E1 -21723.501,E2 -21723.501} C_VEL
LIN {X 0,Y 212.873,Z 720.321,A -85,B 0,C 180,E1 -21726.128,E2 -21726.128} C_VEL
LIN {X 0,Y 212.434,Z 711.537,A -85,B 0,C 180,E1 -21728.466,E2 -21728.466} C_VEL
LIN {X 0,Y 211.167,Z 703.64,A -85,B 0,C 180,E1 -21730.678,E2 -21730.678} C_VEL
LIN {X 0,Y 209.627,Z 697.99,A -85,B 0,C 180,E1 -21732.474,E2 -21732.474} C_VEL
LIN {X 0,Y 207.279,Z 692.306,A -85,B 0,C 180,E1 -21734.6,E2 -21734.6} C_VEL
LIN {X 0,Y 205.587,Z 688.153,A -85,B 0,C 180,E1 -21736.251,E2 -21736.251} C_VEL
LIN {X 0,Y 203.198,Z 684.202,A -85,B 0,C 180,E1 -21738.256,E2 -21738.256} C_VEL
LIN {X 0,Y 202.446,Z 682.357,A -85,B 0,C 180,E1 -21739.077,E2 -21739.077} C_VEL
LIN {X 0,Y 199.856,Z 678.745,A -85,B 0,C 180,E1 -21741.458,E2 -21741.458} C_VEL
LIN {X 0,Y 198.767,Z 675.986,A -85,B 0,C 180,E1 -21742.846,E2 -21742.846} C_VEL
LIN {X 0,Y 195.592,Z 672.424,A -85,B 0,C 180,E1 -21746.515,E2 -21746.515} C_VEL
LIN {X 0,Y 194.097,Z 668.76,A -85,B 0,C 180,E1 -21749.541,E2 -21749.541} C_VEL
LIN {X 0,Y 193.959,Z 667.733,A -85,B 0,C 180,E1 -21754.227,E2 -21754.227} C_VEL
LIN {X 0,Y 193.887,Z 667.146,A -85,B 0,C 180,E1 -21758.747,E2 -21758.747} C_VEL
LIN {X 0,Y 193.976,Z 666.921,A -85,B 0,C 180,E1 -21763.151,E2 -21763.151} C_VEL
LIN {X 0,Y 194.036,Z 667.077,A -85,B 0,C 180,E1 -21765.715,E2 -21765.715} C_VEL
LIN {X 0,Y 195.121,Z 669.379,A -85,B 0,C 180,E1 -21767.858,E2 -21767.858} C_VEL
LIN {X 0,Y 198.339,Z 672.398,A -85,B 0,C 180,E1 -21771.852,E2 -21771.852} C_VEL
LIN {X 0,Y 198.937,Z 672.995,A -85,B 0,C 180,E1 -21772.476,E2 -21772.476} C_VEL
LIN {X 0,Y 200.615,Z 676.254,A -85,B 0,C 180,E1 -21774.472,E2 -21774.472} C_VEL
LIN {X 0,Y 202.996,Z 678.746,A -85,B 0,C 180,E1 -21776.527,E2 -21776.527} C_VEL
LIN {X 0,Y 204.527,Z 681.668,A -85,B 0,C 180,E1 -21778.031,E2 -21778.031} C_VEL
LIN {X 0,Y 205.859,Z 683.494,A -85,B 0,C 180,E1 -21779.096,E2 -21779.096} C_VEL
LIN {X 0,Y 209.714,Z 691.804,A -85,B 0,C 180,E1 -21782.663,E2 -21782.663} C_VEL
LIN {X 0,Y 211.996,Z 698.271,A -85,B 0,C 180,E1 -21785.026,E2 -21785.026} C_VEL
LIN {X 0,Y 213.891,Z 707.9,A -85,B 0,C 180,E1 -21788.027,E2 -21788.027} C_VEL
LIN {X 0,Y 214.609,Z 717.017,A -85,B 0,C 180,E1 -21790.751,E2 -21790.751} C_VEL
LIN {X 0,Y 214.385,Z 723.842,A -85,B 0,C 180,E1 -21792.784,E2 -21792.784} C_VEL
LIN {X 0,Y 213.96,Z 725.754,A -85,B 0,C 180,E1 -21793.293,E2 -21793.293} C_VEL
LIN {X 0,Y 209.989,Z 734.646,A -85,B 0,C 180,E1 -21795.53,E2 -21795.53} C_VEL
LIN {X 0,Y 205.478,Z 743.733,A -85,B 0,C 180,E1 -21798.444,E2 -21798.444} C_VEL
LIN {X 0,Y 201.527,Z 751.025,A -85,B 0,C 180,E1 -21801.535,E2 -21801.535} C_VEL
LIN {X 0,Y 198.583,Z 756.094,A -85,B 0,C 180,E1 -21804.309,E2 -21804.309} C_VEL
LIN {X 0,Y 195.537,Z 760.965,A -85,B 0,C 180,E1 -21807.856,E2 -21807.856} C_VEL
LIN {X 0,Y 193.763,Z 763.649,A -85,B 0,C 180,E1 -21810.517,E2 -21810.517} C_VEL
LIN {X 0,Y 192.359,Z 765.638,A -85,B 0,C 180,E1 -21813.233,E2 -21813.233} C_VEL
LIN {X 0,Y 191.26,Z 766.94,A -85,B 0,C 180,E1 -21816.058,E2 -21816.058} C_VEL
LIN {X 0,Y 190.43,Z 767.572,A -85,B 0,C 180,E1 -21819.192,E2 -21819.192} C_VEL
LIN {X 0,Y 189.971,Z 767.371,A -85,B 0,C 180,E1 -21822.276,E2 -21822.276} C_VEL
LIN {X 0,Y 189.824,Z 766.368,A -85,B 0,C 180,E1 -21825.295,E2 -21825.295} C_VEL
LIN {X 0,Y 189.998,Z 764.568,A -85,B 0,C 180,E1 -21828.254,E2 -21828.254} C_VEL
LIN {X 0,Y 190.387,Z 762.041,A -85,B 0,C 180,E1 -21831.13,E2 -21831.13} C_VEL
LIN {X 0,Y 190.977,Z 758.606,A -85,B 0,C 180,E1 -21834.058,E2 -21834.058} C_VEL
LIN {X 0,Y 191.966,Z 753.541,A -85,B 0,C 180,E1 -21837.357,E2 -21837.357} C_VEL
LIN {X 0,Y 193.464,Z 746.984,A -85,B 0,C 180,E1 -21840.675,E2 -21840.675} C_VEL
LIN {X 0,Y 195.191,Z 739.704,A -85,B 0,C 180,E1 -21843.6,E2 -21843.6} C_VEL
LIN {X 0,Y 197.216,Z 731.105,A -85,B 0,C 180,E1 -21846.364,E2 -21846.364} C_VEL
LIN {X 0,Y 199.522,Z 721.484,A -85,B 0,C 180,E1 -21848.835,E2 -21848.835} C_VEL
LIN {X 0,Y 201.817,Z 710.145,A -85,B 0,C 180,E1 -21851.17,E2 -21851.17} C_VEL
LIN {X 0,Y 200.367,Z 698.283,A -85,B 0,C 180,E1 -21853.441,E2 -21853.441} C_VEL
LIN {X 0,Y 198.291,Z 686.481,A -85,B 0,C 180,E1 -21855.372,E2 -21855.372} C_VEL
LIN {X 0,Y 195.497,Z 674.045,A -85,B 0,C 180,E1 -21857.081,E2 -21857.081} C_VEL
LIN {X 0,Y 192.373,Z 662.625,A -85,B 0,C 180,E1 -21858.441,E2 -21858.441} C_VEL
LIN {X 0,Y 193.007,Z 660.442,A -85,B 0,C 180,E1 -21861.624,E2 -21861.624} C_VEL
LIN {X 0,Y 193.265,Z 660.407,A -85,B 0,C 180,E1 -21867.915,E2 -21867.915} C_VEL
LIN {X 0,Y 193.446,Z 660.388,A -85,B 0,C 180,E1 -21869.999,E2 -21869.999} C_VEL
LIN {X 0,Y 192.953,Z 660.447,A -85,B 0,C 180,E1 -21874.177,E2 -21874.177} C_VEL
LIN {X 0,Y 192.827,Z 660.459,A -85,B 0,C 180,E1 -21878.382,E2 -21878.382} C_VEL
LIN {X 0,Y 192.55,Z 660.537,A -85,B 0,C 180,E1 -21880.713,E2 -21880.713} C_VEL
LIN {X 0,Y 196.069,Z 674.758,A -85,B 0,C 180,E1 -21882.287,E2 -21882.287} C_VEL
LIN {X 0,Y 198.438,Z 686.043,A -85,B 0,C 180,E1 -21883.814,E2 -21883.814} C_VEL
LIN {X 0,Y 200.447,Z 698.427,A -85,B 0,C 180,E1 -21885.816,E2 -21885.816} C_VEL
LIN {X 0,Y 201.764,Z 709.856,A -85,B 0,C 180,E1 -21888.006,E2 -21888.006} C_VEL
LIN {X 0,Y 199.505,Z 720.568,A -85,B 0,C 180,E1 -21890.178,E2 -21890.178} C_VEL
LIN {X 0,Y 197.282,Z 730.244,A -85,B 0,C 180,E1 -21892.65,E2 -21892.65} C_VEL
LIN {X 0,Y 195.008,Z 739.554,A -85,B 0,C 180,E1 -21895.624,E2 -21895.624} C_VEL
LIN {X 0,Y 193.284,Z 746.96,A -85,B 0,C 180,E1 -21898.639,E2 -21898.639} C_VEL
LIN {X 0,Y 191.952,Z 752.85,A -85,B 0,C 180,E1 -21901.635,E2 -21901.635} C_VEL
LIN {X 0,Y 190.996,Z 757.513,A -85,B 0,C 180,E1 -21904.621,E2 -21904.621} C_VEL
LIN {X 0,Y 190.295,Z 761.073,A -85,B 0,C 180,E1 -21907.543,E2 -21907.543} C_VEL
LIN {X 0,Y 189.852,Z 763.68,A -85,B 0,C 180,E1 -21910.375,E2 -21910.375} C_VEL
LIN {X 0,Y 189.732,Z 764.926,A -85,B 0,C 180,E1 -21912.197,E2 -21912.197} C_VEL
LIN {X 0,Y 189.764,Z 766.362,A -85,B 0,C 180,E1 -21915.277,E2 -21915.277} C_VEL
LIN {X 0,Y 190.059,Z 766.929,A -85,B 0,C 180,E1 -21918.271,E2 -21918.271} C_VEL
LIN {X 0,Y 190.628,Z 766.737,A -85,B 0,C 180,E1 -21921.189,E2 -21921.189} C_VEL
LIN {X 0,Y 191.569,Z 765.83,A -85,B 0,C 180,E1 -21924.056,E2 -21924.056} C_VEL
LIN {X 0,Y 193.58,Z 763.084,A -85,B 0,C 180,E1 -21928.278,E2 -21928.278} C_VEL
LIN {X 0,Y 195.413,Z 760.174,A -85,B 0,C 180,E1 -21931.159,E2 -21931.159} C_VEL
LIN {X 0,Y 198.564,Z 754.99,A -85,B 0,C 180,E1 -21934.866,E2 -21934.866} C_VEL
LIN {X 0,Y 202.334,Z 748.256,A -85,B 0,C 180,E1 -21938.323,E2 -21938.323} C_VEL
LIN {X 0,Y 205.798,Z 741.576,A -85,B 0,C 180,E1 -21940.965,E2 -21940.965} C_VEL
LIN {X 0,Y 210.06,Z 732.618,A -85,B 0,C 180,E1 -21943.728,E2 -21943.728} C_VEL
LIN {X 0,Y 213.952,Z 723.34,A -85,B 0,C 180,E1 -21945.98,E2 -21945.98} C_VEL
LIN {X 0,Y 214.408,Z 715.58,A -85,B 0,C 180,E1 -21948.178,E2 -21948.178} C_VEL
LIN {X 0,Y 214.006,Z 707.069,A -85,B 0,C 180,E1 -21950.549,E2 -21950.549} C_VEL
LIN {X 0,Y 212.491,Z 697.337,A -85,B 0,C 180,E1 -21953.33,E2 -21953.33} C_VEL
LIN {X 0,Y 210.693,Z 691.418,A -85,B 0,C 180,E1 -21955.254,E2 -21955.254} C_VEL
LIN {X 0,Y 207.494,Z 684.04,A -85,B 0,C 180,E1 -21958.059,E2 -21958.059} C_VEL
LIN {X 0,Y 205.246,Z 679.354,A -85,B 0,C 180,E1 -21960,E2 -21960} C_VEL
LIN {X 0,Y 202.94,Z 675.477,A -85,B 0,C 180,E1 -21961.93,E2 -21961.93} C_VEL
LIN {X 0,Y 202.209,Z 674.358,A -85,B 0,C 180,E1 -21962.562,E2 -21962.562} C_VEL
LIN {X 0,Y 199.45,Z 671.232,A -85,B 0,C 180,E1 -21964.864,E2 -21964.864} C_VEL
LIN {X 0,Y 198.162,Z 668.872,A -85,B 0,C 180,E1 -21966.239,E2 -21966.239} C_VEL
LIN {X 0,Y 193.832,Z 663.709,A -85,B 0,C 180,E1 -21971.258,E2 -21971.258} C_VEL
LIN {X 0,Y 193.465,Z 662.938,A -85,B 0,C 180,E1 -21972.07,E2 -21972.07} C_VEL
LIN {X 0,Y 193.317,Z 662.398,A -85,B 0,C 180,E1 -21974.743,E2 -21974.743} C_VEL
LIN {X 0,Y 193.036,Z 661.901,A -85,B 0,C 180,E1 -21979.127,E2 -21979.127} C_VEL
LIN {X 0,Y 193.03,Z 662.075,A -85,B 0,C 180,E1 -21984.467,E2 -21984.467} C_VEL
LIN {X 0,Y 193.362,Z 662.751,A -85,B 0,C 180,E1 -21988.197,E2 -21988.197} C_VEL
LIN {X 0,Y 193.706,Z 664.251,A -85,B 0,C 180,E1 -21992.468,E2 -21992.468} C_VEL
LIN {X 0,Y 197.519,Z 669.729,A -85,B 0,C 180,E1 -21997.076,E2 -21997.076} C_VEL
LIN {X 0,Y 198.983,Z 671.265,A -85,B 0,C 180,E1 -21998.419,E2 -21998.419} C_VEL
LIN {X 0,Y 201.409,Z 675.162,A -85,B 0,C 180,E1 -22000.616,E2 -22000.616} C_VEL
LIN {X 0,Y 203.082,Z 677.428,A -85,B 0,C 180,E1 -22001.939,E2 -22001.939} C_VEL
LIN {X 0,Y 205.53,Z 681.878,A -85,B 0,C 180,E1 -22003.928,E2 -22003.928} C_VEL
LIN {X 0,Y 209.329,Z 689.615,A -85,B 0,C 180,E1 -22006.906,E2 -22006.906} C_VEL
LIN {X 0,Y 210.973,Z 695.186,A -85,B 0,C 180,E1 -22008.548,E2 -22008.548} C_VEL
LIN {X 0,Y 212.344,Z 705.257,A -85,B 0,C 180,E1 -22011.036,E2 -22011.036} C_VEL
LIN {X 0,Y 212.735,Z 715.619,A -85,B 0,C 180,E1 -22013.513,E2 -22013.513} C_VEL
LIN {X 0,Y 212.125,Z 725.411,A -85,B 0,C 180,E1 -22015.923,E2 -22015.923} C_VEL
LIN {X 0,Y 211.078,Z 732.684,A -85,B 0,C 180,E1 -22017.811,E2 -22017.811} C_VEL
LIN {X 0,Y 209.629,Z 738.518,A -85,B 0,C 180,E1 -22019.391,E2 -22019.391} C_VEL
LIN {X 0,Y 205.621,Z 747.575,A -85,B 0,C 180,E1 -22021.969,E2 -22021.969} C_VEL
LIN {X 0,Y 201.73,Z 755.345,A -85,B 0,C 180,E1 -22024.738,E2 -22024.738} C_VEL
LIN {X 0,Y 200.662,Z 757.357,A -85,B 0,C 180,E1 -22025.589,E2 -22025.589} C_VEL
LIN {X 0,Y 198.459,Z 760.43,A -85,B 0,C 180,E1 -22026.904,E2 -22026.904} C_VEL
LIN {X 0,Y 193.394,Z 764.967,A -85,B 0,C 180,E1 -22029.022,E2 -22029.022} C_VEL
LIN {X 0,Y 188.567,Z 768.812,A -85,B 0,C 180,E1 -22031.349,E2 -22031.349} C_VEL
LIN {X 0,Y 186.785,Z 770.735,A -85,B 0,C 180,E1 -22032.964,E2 -22032.964} C_VEL
LIN {X 0,Y 184.812,Z 774.061,A -85,B 0,C 180,E1 -22036.812,E2 -22036.812} C_VEL
LIN {X 0,Y 183.52,Z 776.28,A -85,B 0,C 180,E1 -22041.19,E2 -22041.19} C_VEL
LIN {X 0,Y 183.118,Z 776.882,A -85,B 0,C 180,E1 -22045.599,E2 -22045.599} C_VEL
LIN {X 0,Y 183.165,Z 776.582,A -85,B 0,C 180,E1 -22048.627,E2 -22048.627} C_VEL
LIN {X 0,Y 183.255,Z 777.252,A -85,B 0,C 180,E1 -22050.001,E2 -22050.001} C_VEL
LIN {X 0,Y 183.078,Z 778.218,A -85,B 0,C 180,E1 -22054.404,E2 -22054.404} C_VEL
LIN {X 0,Y 183.546,Z 777.66,A -85,B 0,C 180,E1 -22058.811,E2 -22058.811} C_VEL
LIN {X 0,Y 184.835,Z 775.514,A -85,B 0,C 180,E1 -22063.188,E2 -22063.188} C_VEL
LIN {X 0,Y 187.113,Z 771.81,A -85,B 0,C 180,E1 -22067.487,E2 -22067.487} C_VEL
LIN {X 0,Y 189.683,Z 767.881,A -85,B 0,C 180,E1 -22070.61,E2 -22070.61} C_VEL
LIN {X 0,Y 192.604,Z 762.898,A -85,B 0,C 180,E1 -22073.665,E2 -22073.665} C_VEL
LIN {X 0,Y 196.043,Z 756.743,A -85,B 0,C 180,E1 -22076.624,E2 -22076.624} C_VEL
LIN {X 0,Y 200.16,Z 749.194,A -85,B 0,C 180,E1 -22079.444,E2 -22079.444} C_VEL
LIN {X 0,Y 204.653,Z 739.909,A -85,B 0,C 180,E1 -22082.161,E2 -22082.161} C_VEL
LIN {X 0,Y 206.412,Z 731.678,A -85,B 0,C 180,E1 -22084.571,E2 -22084.571} C_VEL
LIN {X 0,Y 207.245,Z 722.151,A -85,B 0,C 180,E1 -22087.289,E2 -22087.289} C_VEL
LIN {X 0,Y 206.99,Z 713.441,A -85,B 0,C 180,E1 -22089.785,E2 -22089.785} C_VEL
LIN {X 0,Y 206.104,Z 706.598,A -85,B 0,C 180,E1 -22091.883,E2 -22091.883} C_VEL
LIN {X 0,Y 204.562,Z 701.216,A -85,B 0,C 180,E1 -22093.823,E2 -22093.823} C_VEL
LIN {X 0,Y 201.714,Z 693.59,A -85,B 0,C 180,E1 -22097.027,E2 -22097.027} C_VEL
LIN {X 0,Y 199.108,Z 688.241,A -85,B 0,C 180,E1 -22099.815,E2 -22099.815} C_VEL
LIN {X 0,Y 196.625,Z 683.987,A -85,B 0,C 180,E1 -22102.581,E2 -22102.581} C_VEL
LIN {X 0,Y 195.638,Z 681.918,A -85,B 0,C 180,E1 -22103.967,E2 -22103.967} C_VEL
LIN {X 0,Y 193.041,Z 678.232,A -85,B 0,C 180,E1 -22107.675,E2 -22107.675} C_VEL
LIN {X 0,Y 192.084,Z 675.457,A -85,B 0,C 180,E1 -22110.007,E2 -22110.007} C_VEL
LIN {X 0,Y 190.265,Z 673.537,A -85,B 0,C 180,E1 -22116.026,E2 -22116.026} C_VEL
LIN {X 0,Y 190.485,Z 673.226,A -85,B 0,C 180,E1 -22120.606,E2 -22120.606} C_VEL
LIN {X 0,Y 192.194,Z 673.854,A -85,B 0,C 180,E1 -22125.304,E2 -22125.304} C_VEL
LIN {X 0,Y 193.293,Z 676.441,A -85,B 0,C 180,E1 -22127.928,E2 -22127.928} C_VEL
LIN {X 0,Y 196.213,Z 679.152,A -85,B 0,C 180,E1 -22131.763,E2 -22131.763} C_VEL
LIN {X 0,Y 197.846,Z 682.619,A -85,B 0,C 180,E1 -22134.066,E2 -22134.066} C_VEL
LIN {X 0,Y 199.819,Z 684.821,A -85,B 0,C 180,E1 -22135.966,E2 -22135.966} C_VEL
LIN {X 0,Y 202.248,Z 689.334,A -85,B 0,C 180,E1 -22138.544,E2 -22138.544} C_VEL
LIN {X 0,Y 205.323,Z 696.784,A -85,B 0,C 180,E1 -22141.962,E2 -22141.962} C_VEL
LIN {X 0,Y 207.337,Z 703.375,A -85,B 0,C 180,E1 -22144.513,E2 -22144.513} C_VEL
LIN {X 0,Y 208.675,Z 713.059,A -85,B 0,C 180,E1 -22147.742,E2 -22147.742} C_VEL
LIN {X 0,Y 208.833,Z 721.143,A -85,B 0,C 180,E1 -22150.332,E2 -22150.332} C_VEL
LIN {X 0,Y 208.373,Z 726.426,A -85,B 0,C 180,E1 -22152.007,E2 -22152.007} C_VEL
LIN {X 0,Y 204.369,Z 735.288,A -85,B 0,C 180,E1 -22154.338,E2 -22154.338} C_VEL
LIN {X 0,Y 200.182,Z 743.236,A -85,B 0,C 180,E1 -22156.927,E2 -22156.927} C_VEL
LIN {X 0,Y 196.392,Z 749.778,A -85,B 0,C 180,E1 -22159.633,E2 -22159.633} C_VEL
LIN {X 0,Y 192.535,Z 756.096,A -85,B 0,C 180,E1 -22163.055,E2 -22163.055} C_VEL
LIN {X 0,Y 189.065,Z 761.21,A -85,B 0,C 180,E1 -22166.856,E2 -22166.856} C_VEL
LIN {X 0,Y 186.841,Z 764.282,A -85,B 0,C 180,E1 -22170.1,E2 -22170.1} C_VEL
LIN {X 0,Y 185.159,Z 766.363,A -85,B 0,C 180,E1 -22173.378,E2 -22173.378} C_VEL
LIN {X 0,Y 183.631,Z 767.736,A -85,B 0,C 180,E1 -22177.761,E2 -22177.761} C_VEL
LIN {X 0,Y 183.058,Z 767.745,A -85,B 0,C 180,E1 -22180.743,E2 -22180.743} C_VEL
LIN {X 0,Y 182.742,Z 767.034,A -85,B 0,C 180,E1 -22183.809,E2 -22183.809} C_VEL
LIN {X 0,Y 182.765,Z 765.528,A -85,B 0,C 180,E1 -22186.939,E2 -22186.939} C_VEL
LIN {X 0,Y 183.298,Z 762.097,A -85,B 0,C 180,E1 -22191.179,E2 -22191.179} C_VEL
LIN {X 0,Y 184.153,Z 757.476,A -85,B 0,C 180,E1 -22195.077,E2 -22195.077} C_VEL
LIN {X 0,Y 185.27,Z 752,A -85,B 0,C 180,E1 -22198.52,E2 -22198.52} C_VEL
LIN {X 0,Y 186.959,Z 744.901,A -85,B 0,C 180,E1 -22201.972,E2 -22201.972} C_VEL
LIN {X 0,Y 189.156,Z 736.218,A -85,B 0,C 180,E1 -22205.291,E2 -22205.291} C_VEL
LIN {X 0,Y 191.52,Z 726.561,A -85,B 0,C 180,E1 -22208.178,E2 -22208.178} C_VEL
LIN {X 0,Y 193.962,Z 716.089,A -85,B 0,C 180,E1 -22210.658,E2 -22210.658} C_VEL
LIN {X 0,Y 194.943,Z 711.342,A -85,B 0,C 180,E1 -22211.611,E2 -22211.611} C_VEL
LIN {X 0,Y 193.936,Z 701.945,A -85,B 0,C 180,E1 -22213.543,E2 -22213.543} C_VEL
LIN {X 0,Y 192.261,Z 691.317,A -85,B 0,C 180,E1 -22215.444,E2 -22215.444} C_VEL
LIN {X 0,Y 189.721,Z 679.018,A -85,B 0,C 180,E1 -22217.322,E2 -22217.322} C_VEL
LIN {X 0,Y 186.104,Z 665.486,A -85,B 0,C 180,E1 -22219.072,E2 -22219.072} C_VEL
LIN {X 0,Y 185.442,Z 662.841,A -85,B 0,C 180,E1 -22219.387,E2 -22219.387} C_VEL
LIN {X 0,Y 185.95,Z 661.32,A -85,B 0,C 180,E1 -22221.851,E2 -22221.851} C_VEL
LIN {X 0,Y 186.209,Z 661.286,A -85,B 0,C 180,E1 -22227.836,E2 -22227.836} C_VEL
LIN {X 0,Y 186.409,Z 661.264,A -85,B 0,C 180,E1 -22229.999,E2 -22229.999} C_VEL
LIN {X 0,Y 185.895,Z 661.326,A -85,B 0,C 180,E1 -22234.335,E2 -22234.335} C_VEL
LIN {X 0,Y 185.746,Z 661.343,A -85,B 0,C 180,E1 -22238.704,E2 -22238.704} C_VEL
LIN {X 0,Y 185.648,Z 661.443,A -85,B 0,C 180,E1 -22239.809,E2 -22239.809} C_VEL
LIN {X 0,Y 188.797,Z 673.241,A -85,B 0,C 180,E1 -22241.193,E2 -22241.193} C_VEL
LIN {X 0,Y 191.548,Z 686.115,A -85,B 0,C 180,E1 -22242.988,E2 -22242.988} C_VEL
LIN {X 0,Y 193.487,Z 698.204,A -85,B 0,C 180,E1 -22244.998,E2 -22244.998} C_VEL
LIN {X 0,Y 194.842,Z 709.879,A -85,B 0,C 180,E1 -22247.311,E2 -22247.311} C_VEL
LIN {X 0,Y 194.5,Z 712.743,A -85,B 0,C 180,E1 -22247.886,E2 -22247.886} C_VEL
LIN {X 0,Y 191.97,Z 723.827,A -85,B 0,C 180,E1 -22250.351,E2 -22250.351} C_VEL
LIN {X 0,Y 189.601,Z 733.673,A -85,B 0,C 180,E1 -22253.152,E2 -22253.152} C_VEL
LIN {X 0,Y 187.402,Z 742.433,A -85,B 0,C 180,E1 -22256.299,E2 -22256.299} C_VEL
LIN {X 0,Y 185.697,Z 749.444,A -85,B 0,C 180,E1 -22259.486,E2 -22259.486} C_VEL
LIN {X 0,Y 184.356,Z 755.462,A -85,B 0,C 180,E1 -22262.999,E2 -22262.999} C_VEL
LIN {X 0,Y 183.447,Z 759.98,A -85,B 0,C 180,E1 -22266.435,E2 -22266.435} C_VEL
LIN {X 0,Y 182.702,Z 764.062,A -85,B 0,C 180,E1 -22270.838,E2 -22270.838} C_VEL
LIN {X 0,Y 182.632,Z 765.851,A -85,B 0,C 180,E1 -22273.84,E2 -22273.84} C_VEL
LIN {X 0,Y 182.774,Z 766.882,A -85,B 0,C 180,E1 -22276.934,E2 -22276.934} C_VEL
LIN {X 0,Y 183.28,Z 767.144,A -85,B 0,C 180,E1 -22280.076,E2 -22280.076} C_VEL
LIN {X 0,Y 184.143,Z 766.595,A -85,B 0,C 180,E1 -22283.27,E2 -22283.27} C_VEL
LIN {X 0,Y 185.457,Z 765.196,A -85,B 0,C 180,E1 -22286.479,E2 -22286.479} C_VEL
LIN {X 0,Y 187.239,Z 762.884,A -85,B 0,C 180,E1 -22289.687,E2 -22289.687} C_VEL
LIN {X 0,Y 190.165,Z 758.54,A -85,B 0,C 180,E1 -22293.673,E2 -22293.673} C_VEL
LIN {X 0,Y 193.436,Z 753.424,A -85,B 0,C 180,E1 -22297.01,E2 -22297.01} C_VEL
LIN {X 0,Y 197.307,Z 746.856,A -85,B 0,C 180,E1 -22300.234,E2 -22300.234} C_VEL
LIN {X 0,Y 201.141,Z 739.809,A -85,B 0,C 180,E1 -22302.909,E2 -22302.909} C_VEL
LIN {X 0,Y 205.391,Z 731.221,A -85,B 0,C 180,E1 -22305.468,E2 -22305.468} C_VEL
LIN {X 0,Y 207.949,Z 725.558,A -85,B 0,C 180,E1 -22306.863,E2 -22306.863} C_VEL
LIN {X 0,Y 208.635,Z 718.949,A -85,B 0,C 180,E1 -22308.832,E2 -22308.832} C_VEL
LIN {X 0,Y 208.605,Z 710.811,A -85,B 0,C 180,E1 -22311.28,E2 -22311.28} C_VEL
LIN {X 0,Y 207.541,Z 701.398,A -85,B 0,C 180,E1 -22314.169,E2 -22314.169} C_VEL
LIN {X 0,Y 206.077,Z 695.932,A -85,B 0,C 180,E1 -22316.089,E2 -22316.089} C_VEL
LIN {X 0,Y 203.244,Z 688.843,A -85,B 0,C 180,E1 -22319.029,E2 -22319.029} C_VEL
LIN {X 0,Y 201.23,Z 684.324,A -85,B 0,C 180,E1 -22321.094,E2 -22321.094} C_VEL
LIN {X 0,Y 199.285,Z 680.614,A -85,B 0,C 180,E1 -22323.042,E2 -22323.042} C_VEL
LIN {X 0,Y 196.656,Z 677.267,A -85,B 0,C 180,E1 -22325.583,E2 -22325.583} C_VEL
LIN {X 0,Y 195.634,Z 675.271,A -85,B 0,C 180,E1 -22326.838,E2 -22326.838} C_VEL
LIN {X 0,Y 191.959,Z 670.254,A -85,B 0,C 180,E1 -22331.838,E2 -22331.838} C_VEL
LIN {X 0,Y 191.442,Z 669.577,A -85,B 0,C 180,E1 -22332.725,E2 -22332.725} C_VEL
LIN {X 0,Y 189.008,Z 667.741,A -85,B 0,C 180,E1 -22338.572,E2 -22338.572} C_VEL
LIN {X 0,Y 188.791,Z 667.72,A -85,B 0,C 180,E1 -22344.173,E2 -22344.173} C_VEL
LIN {X 0,Y 190.349,Z 669.507,A -85,B 0,C 180,E1 -22349.228,E2 -22349.228} C_VEL
LIN {X 0,Y 192.066,Z 671.258,A -85,B 0,C 180,E1 -22352.208,E2 -22352.208} C_VEL
LIN {X 0,Y 195.574,Z 676.55,A -85,B 0,C 180,E1 -22356.858,E2 -22356.858} C_VEL
LIN {X 0,Y 196.557,Z 677.771,A -85,B 0,C 180,E1 -22357.874,E2 -22357.874} C_VEL
LIN {X 0,Y 199.089,Z 681.969,A -85,B 0,C 180,E1 -22360.44,E2 -22360.44} C_VEL
LIN {X 0,Y 202.757,Z 689.13,A -85,B 0,C 180,E1 -22363.888,E2 -22363.888} C_VEL
LIN {X 0,Y 205.068,Z 694.38,A -85,B 0,C 180,E1 -22366.03,E2 -22366.03} C_VEL
LIN {X 0,Y 206.364,Z 699.441,A -85,B 0,C 180,E1 -22367.648,E2 -22367.648} C_VEL
LIN {X 0,Y 207.28,Z 710.401,A -85,B 0,C 180,E1 -22370.522,E2 -22370.522} C_VEL
LIN {X 0,Y 207.09,Z 720.135,A -85,B 0,C 180,E1 -22373.03,E2 -22373.03} C_VEL
LIN {X 0,Y 205.798,Z 730.841,A -85,B 0,C 180,E1 -22375.895,E2 -22375.895} C_VEL
LIN {X 0,Y 203.764,Z 739.171,A -85,B 0,C 180,E1 -22378.267,E2 -22378.267} C_VEL
LIN {X 0,Y 199.443,Z 748.436,A -85,B 0,C 180,E1 -22381.02,E2 -22381.02} C_VEL
LIN {X 0,Y 195.381,Z 755.967,A -85,B 0,C 180,E1 -22383.856,E2 -22383.856} C_VEL
LIN {X 0,Y 192.439,Z 761.152,A -85,B 0,C 180,E1 -22386.315,E2 -22386.315} C_VEL
LIN {X 0,Y 189.616,Z 766.252,A -85,B 0,C 180,E1 -22389.385,E2 -22389.385} C_VEL
LIN {X 0,Y 186.785,Z 770.735,A -85,B 0,C 180,E1 -22392.964,E2 -22392.964} C_VEL
LIN {X 0,Y 185.131,Z 772.426,A -85,B 0,C 180,E1 -22394.64,E2 -22394.64} C_VEL
LIN {X 0,Y 180.999,Z 774.622,A -85,B 0,C 180,E1 -22397.383,E2 -22397.383} C_VEL
LIN {X 0,Y 177.855,Z 775.773,A -85,B 0,C 180,E1 -22399.685,E2 -22399.685} C_VEL
LIN {X 0,Y 176.43,Z 776.333,A -85,B 0,C 180,E1 -22401.534,E2 -22401.534} C_VEL
LIN {X 0,Y 176.251,Z 776.42,A -85,B 0,C 180,E1 -22402.171,E2 -22402.171} C_VEL
LIN {X 0,Y 176.016,Z 776.535,A -85,B 0,C 180,E1 -22406.569,E2 -22406.569} C_VEL
LIN {X 0,Y 176.075,Z 776.182,A -85,B 0,C 180,E1 -22408.571,E2 -22408.571} C_VEL
LIN {X 0,Y 176.176,Z 776.864,A -85,B 0,C 180,E1 -22410.001,E2 -22410.001} C_VEL
LIN {X 0,Y 175.991,Z 777.816,A -85,B 0,C 180,E1 -22413.292,E2 -22413.292} C_VEL
LIN {X 0,Y 176.154,Z 777.937,A -85,B 0,C 180,E1 -22416.875,E2 -22416.875} C_VEL
LIN {X 0,Y 177.08,Z 776.743,A -85,B 0,C 180,E1 -22421.447,E2 -22421.447} C_VEL
LIN {X 0,Y 177.913,Z 775.556,A -85,B 0,C 180,E1 -22423.711,E2 -22423.711} C_VEL
LIN {X 0,Y 178.951,Z 773.962,A -85,B 0,C 180,E1 -22425.958,E2 -22425.958} C_VEL
LIN {X 0,Y 181.212,Z 770.82,A -85,B 0,C 180,E1 -22429.249,E2 -22429.249} C_VEL
LIN {X 0,Y 185.137,Z 765.095,A -85,B 0,C 180,E1 -22433.491,E2 -22433.491} C_VEL
LIN {X 0,Y 188.459,Z 759.539,A -85,B 0,C 180,E1 -22436.584,E2 -22436.584} C_VEL
LIN {X 0,Y 192.545,Z 752.682,A -85,B 0,C 180,E1 -22439.523,E2 -22439.523} C_VEL
LIN {X 0,Y 197.193,Z 744.226,A -85,B 0,C 180,E1 -22442.318,E2 -22442.318} C_VEL
LIN {X 0,Y 198.72,Z 741.05,A -85,B 0,C 180,E1 -22443.243,E2 -22443.243} C_VEL
LIN {X 0,Y 200.65,Z 733.264,A -85,B 0,C 180,E1 -22445.693,E2 -22445.693} C_VEL
LIN {X 0,Y 201.621,Z 725.022,A -85,B 0,C 180,E1 -22448.206,E2 -22448.206} C_VEL
LIN {X 0,Y 201.742,Z 716.608,A -85,B 0,C 180,E1 -22450.801,E2 -22450.801} C_VEL
LIN {X 0,Y 200.997,Z 709.617,A -85,B 0,C 180,E1 -22453.153,E2 -22453.153} C_VEL
LIN {X 0,Y 199.254,Z 703.276,A -85,B 0,C 180,E1 -22455.753,E2 -22455.753} C_VEL
LIN {X 0,Y 197.892,Z 699.322,A -85,B 0,C 180,E1 -22457.564,E2 -22457.564} C_VEL
LIN {X 0,Y 196.098,Z 695.184,A -85,B 0,C 180,E1 -22459.826,E2 -22459.826} C_VEL
LIN {X 0,Y 192.911,Z 688.352,A -85,B 0,C 180,E1 -22464.345,E2 -22464.345} C_VEL
LIN {X 0,Y 190.31,Z 683.914,A -85,B 0,C 180,E1 -22468.868,E2 -22468.868} C_VEL
LIN {X 0,Y 190.057,Z 682.982,A -85,B 0,C 180,E1 -22469.654,E2 -22469.654} C_VEL
LIN {X 0,Y 189.565,Z 681.834,A -85,B 0,C 180,E1 -22471.186,E2 -22471.186} C_VEL
LIN {X 0,Y 188.296,Z 680.239,A -85,B 0,C 180,E1 -22476.879,E2 -22476.879} C_VEL
LIN {X 0,Y 189.101,Z 680.226,A -85,B 0,C 180,E1 -22482.703,E2 -22482.703} C_VEL
LIN {X 0,Y 190.018,Z 680.629,A -85,B 0,C 180,E1 -22484.995,E2 -22484.995} C_VEL
LIN {X 0,Y 190.729,Z 682.72,A -85,B 0,C 180,E1 -22487.227,E2 -22487.227} C_VEL
LIN {X 0,Y 193.551,Z 686.086,A -85,B 0,C 180,E1 -22491.649,E2 -22491.649} C_VEL
LIN {X 0,Y 194.928,Z 689.027,A -85,B 0,C 180,E1 -22493.791,E2 -22493.791} C_VEL
LIN {X 0,Y 196.72,Z 691.683,A -85,B 0,C 180,E1 -22495.903,E2 -22495.903} C_VEL
LIN {X 0,Y 198.418,Z 694.987,A -85,B 0,C 180,E1 -22497.97,E2 -22497.97} C_VEL
LIN {X 0,Y 200.981,Z 702.099,A -85,B 0,C 180,E1 -22501.431,E2 -22501.431} C_VEL
LIN {X 0,Y 202.26,Z 706.988,A -85,B 0,C 180,E1 -22503.486,E2 -22503.486} C_VEL
LIN {X 0,Y 203.114,Z 715.174,A -85,B 0,C 180,E1 -22506.457,E2 -22506.457} C_VEL
LIN {X 0,Y 203.146,Z 722.432,A -85,B 0,C 180,E1 -22508.956,E2 -22508.956} C_VEL
LIN {X 0,Y 202.678,Z 727.361,A -85,B 0,C 180,E1 -22510.65,E2 -22510.65} C_VEL
LIN {X 0,Y 202.267,Z 729.156,A -85,B 0,C 180,E1 -22511.22,E2 -22511.22} C_VEL
LIN {X 0,Y 198.433,Z 736.71,A -85,B 0,C 180,E1 -22513.31,E2 -22513.31} C_VEL
LIN {X 0,Y 194.404,Z 743.87,A -85,B 0,C 180,E1 -22515.731,E2 -22515.731} C_VEL
LIN {X 0,Y 189.767,Z 751.341,A -85,B 0,C 180,E1 -22518.993,E2 -22518.993} C_VEL
LIN {X 0,Y 186.087,Z 756.84,A -85,B 0,C 180,E1 -22522.19,E2 -22522.19} C_VEL
LIN {X 0,Y 182.488,Z 761.714,A -85,B 0,C 180,E1 -22526.022,E2 -22526.022} C_VEL
LIN {X 0,Y 180.248,Z 764.508,A -85,B 0,C 180,E1 -22529.111,E2 -22529.111} C_VEL
LIN {X 0,Y 177.798,Z 767.184,A -85,B 0,C 180,E1 -22533.891,E2 -22533.891} C_VEL
LIN {X 0,Y 176.64,Z 767.995,A -85,B 0,C 180,E1 -22537.273,E2 -22537.273} C_VEL
LIN {X 0,Y 175.969,Z 767.927,A -85,B 0,C 180,E1 -22540.637,E2 -22540.637} C_VEL
LIN {X 0,Y 175.635,Z 767.056,A -85,B 0,C 180,E1 -22543.922,E2 -22543.922} C_VEL
LIN {X 0,Y 175.674,Z 765.421,A -85,B 0,C 180,E1 -22547.147,E2 -22547.147} C_VEL
LIN {X 0,Y 176.034,Z 763.04,A -85,B 0,C 180,E1 -22550.298,E2 -22550.298} C_VEL
LIN {X 0,Y 176.591,Z 759.901,A -85,B 0,C 180,E1 -22553.346,E2 -22553.346} C_VEL
LIN {X 0,Y 177.624,Z 754.919,A -85,B 0,C 180,E1 -22557.04,E2 -22557.04} C_VEL
LIN {X 0,Y 179.225,Z 747.915,A -85,B 0,C 180,E1 -22560.961,E2 -22560.961} C_VEL
LIN {X 0,Y 181.072,Z 740.697,A -85,B 0,C 180,E1 -22564.13,E2 -22564.13} C_VEL
LIN {X 0,Y 183.168,Z 732.428,A -85,B 0,C 180,E1 -22567.052,E2 -22567.052} C_VEL
LIN {X 0,Y 185.699,Z 722.62,A -85,B 0,C 180,E1 -22569.796,E2 -22569.796} C_VEL
LIN {X 0,Y 187.98,Z 712.666,A -85,B 0,C 180,E1 -22572.034,E2 -22572.034} C_VEL
LIN {X 0,Y 187.404,Z 705.214,A -85,B 0,C 180,E1 -22573.664,E2 -22573.664} C_VEL
LIN {X 0,Y 185.701,Z 693.582,A -85,B 0,C 180,E1 -22575.908,E2 -22575.908} C_VEL
LIN {X 0,Y 183.344,Z 681.374,A -85,B 0,C 180,E1 -22577.924,E2 -22577.924} C_VEL
LIN {X 0,Y 180.08,Z 668.778,A -85,B 0,C 180,E1 -22579.707,E2 -22579.707} C_VEL
LIN {X 0,Y 178.602,Z 663.036,A -85,B 0,C 180,E1 -22580.413,E2 -22580.413} C_VEL
LIN {X 0,Y 178.906,Z 662.197,A -85,B 0,C 180,E1 -22581.812,E2 -22581.812} C_VEL
LIN {X 0,Y 179.154,Z 662.165,A -85,B 0,C 180,E1 -22587.751,E2 -22587.751} C_VEL
LIN {X 0,Y 179.372,Z 662.141,A -85,B 0,C 180,E1 -22589.999,E2 -22589.999} C_VEL
LIN {X 0,Y 178.837,Z 662.206,A -85,B 0,C 180,E1 -22594.507,E2 -22594.507} C_VEL
LIN {X 0,Y 178.715,Z 662.219,A -85,B 0,C 180,E1 -22598.764,E2 -22598.764} C_VEL
LIN {X 0,Y 180.295,Z 666.791,A -85,B 0,C 180,E1 -22599.391,E2 -22599.391} C_VEL
LIN {X 0,Y 183.262,Z 679.283,A -85,B 0,C 180,E1 -22601.054,E2 -22601.054} C_VEL
LIN {X 0,Y 185.72,Z 692.318,A -85,B 0,C 180,E1 -22603.122,E2 -22603.122} C_VEL
LIN {X 0,Y 187.268,Z 703.492,A -85,B 0,C 180,E1 -22605.229,E2 -22605.229} C_VEL
LIN {X 0,Y 188.003,Z 711.021,A -85,B 0,C 180,E1 -22606.84,E2 -22606.84} C_VEL
LIN {X 0,Y 185.861,Z 720.988,A -85,B 0,C 180,E1 -22609.032,E2 -22609.032} C_VEL
LIN {X 0,Y 183.255,Z 731.569,A -85,B 0,C 180,E1 -22611.957,E2 -22611.957} C_VEL
LIN {X 0,Y 181.212,Z 739.351,A -85,B 0,C 180,E1 -22614.639,E2 -22614.639} C_VEL
LIN {X 0,Y 179.225,Z 747.274,A -85,B 0,C 180,E1 -22618.069,E2 -22618.069} C_VEL
LIN {X 0,Y 177.738,Z 753.562,A -85,B 0,C 180,E1 -22621.54,E2 -22621.54} C_VEL
LIN {X 0,Y 176.592,Z 758.761,A -85,B 0,C 180,E1 -22625.243,E2 -22625.243} C_VEL
LIN {X 0,Y 175.937,Z 762.053,A -85,B 0,C 180,E1 -22628.345,E2 -22628.345} C_VEL
LIN {X 0,Y 175.629,Z 763.866,A -85,B 0,C 180,E1 -22630.508,E2 -22630.508} C_VEL
LIN {X 0,Y 175.531,Z 765.903,A -85,B 0,C 180,E1 -22633.888,E2 -22633.888} C_VEL
LIN {X 0,Y 175.692,Z 767.029,A -85,B 0,C 180,E1 -22637.154,E2 -22637.154} C_VEL
LIN {X 0,Y 176.223,Z 767.372,A -85,B 0,C 180,E1 -22640.349,E2 -22640.349} C_VEL
LIN {X 0,Y 177.077,Z 766.984,A -85,B 0,C 180,E1 -22643.463,E2 -22643.463} C_VEL
LIN {X 0,Y 178.328,Z 765.843,A -85,B 0,C 180,E1 -22646.513,E2 -22646.513} C_VEL
LIN {X 0,Y 180.847,Z 762.867,A -85,B 0,C 180,E1 -22650.937,E2 -22650.937} C_VEL
LIN {X 0,Y 184.241,Z 758.257,A -85,B 0,C 180,E1 -22655.19,E2 -22655.19} C_VEL
LIN {X 0,Y 188.262,Z 752.368,A -85,B 0,C 180,E1 -22658.947,E2 -22658.947} C_VEL
LIN {X 0,Y 192.156,Z 746.05,A -85,B 0,C 180,E1 -22661.973,E2 -22661.973} C_VEL
LIN {X 0,Y 196.929,Z 737.652,A -85,B 0,C 180,E1 -22665.053,E2 -22665.053} C_VEL
LIN {X 0,Y 201.49,Z 728.61,A -85,B 0,C 180,E1 -22667.586,E2 -22667.586} C_VEL
LIN {X 0,Y 202.165,Z 727.121,A -85,B 0,C 180,E1 -22667.961,E2 -22667.961} C_VEL
LIN {X 0,Y 202.982,Z 720.716,A -85,B 0,C 180,E1 -22670.031,E2 -22670.031} C_VEL
LIN {X 0,Y 203.104,Z 712.177,A -85,B 0,C 180,E1 -22672.787,E2 -22672.787} C_VEL
LIN {X 0,Y 202.557,Z 705.441,A -85,B 0,C 180,E1 -22675.024,E2 -22675.024} C_VEL
LIN {X 0,Y 201.503,Z 700.71,A -85,B 0,C 180,E1 -22676.813,E2 -22676.813} C_VEL
LIN {X 0,Y 198.523,Z 692.401,A -85,B 0,C 180,E1 -22680.554,E2 -22680.554} C_VEL
LIN {X 0,Y 196.456,Z 687.504,A -85,B 0,C 180,E1 -22683.086,E2 -22683.086} C_VEL
LIN {X 0,Y 193.673,Z 683.29,A -85,B 0,C 180,E1 -22686.25,E2 -22686.25} C_VEL
LIN {X 0,Y 192.976,Z 681.65,A -85,B 0,C 180,E1 -22687.323,E2 -22687.323} C_VEL
LIN {X 0,Y 189.552,Z 676.402,A -85,B 0,C 180,E1 -22692.854,E2 -22692.854} C_VEL
LIN {X 0,Y 187.35,Z 674.622,A -85,B 0,C 180,E1 -22698.743,E2 -22698.743} C_VEL
LIN {X 0,Y 187.218,Z 674.697,A -85,B 0,C 180,E1 -22704.389,E2 -22704.389} C_VEL
LIN {X 0,Y 188.714,Z 676.46,A -85,B 0,C 180,E1 -22709.293,E2 -22709.293} C_VEL
LIN {X 0,Y 189.992,Z 677.921,A -85,B 0,C 180,E1 -22711.764,E2 -22711.764} C_VEL
LIN {X 0,Y 192.487,Z 682.346,A -85,B 0,C 180,E1 -22715.746,E2 -22715.746} C_VEL
LIN {X 0,Y 193.619,Z 683.575,A -85,B 0,C 180,E1 -22717.009,E2 -22717.009} C_VEL
LIN {X 0,Y 195.549,Z 687.426,A -85,B 0,C 180,E1 -22719.424,E2 -22719.424} C_VEL
LIN {X 0,Y 196.276,Z 688.412,A -85,B 0,C 180,E1 -22720.13,E2 -22720.13} C_VEL
LIN {X 0,Y 199.345,Z 695.625,A -85,B 0,C 180,E1 -22723.64,E2 -22723.64} C_VEL
LIN {X 0,Y 201.073,Z 700.434,A -85,B 0,C 180,E1 -22725.651,E2 -22725.651} C_VEL
LIN {X 0,Y 201.817,Z 704.55,A -85,B 0,C 180,E1 -22726.995,E2 -22726.995} C_VEL
LIN {X 0,Y 201.987,Z 716.168,A -85,B 0,C 180,E1 -22730.23,E2 -22730.23} C_VEL
LIN {X 0,Y 201.103,Z 725.901,A -85,B 0,C 180,E1 -22732.928,E2 -22732.928} C_VEL
LIN {X 0,Y 199.337,Z 735.282,A -85,B 0,C 180,E1 -22735.661,E2 -22735.661} C_VEL
LIN {X 0,Y 197.174,Z 741.937,A -85,B 0,C 180,E1 -22737.681,E2 -22737.681} C_VEL
LIN {X 0,Y 192.555,Z 750.578,A -85,B 0,C 180,E1 -22740.481,E2 -22740.481} C_VEL
LIN {X 0,Y 188.385,Z 757.669,A -85,B 0,C 180,E1 -22743.406,E2 -22743.406} C_VEL
LIN {X 0,Y 184.992,Z 763.407,A -85,B 0,C 180,E1 -22746.492,E2 -22746.492} C_VEL
LIN {X 0,Y 182.041,Z 767.985,A -85,B 0,C 180,E1 -22749.669,E2 -22749.669} C_VEL
LIN {X 0,Y 179.58,Z 771.518,A -85,B 0,C 180,E1 -22752.932,E2 -22752.932} C_VEL
LIN {X 0,Y 177.89,Z 774.105,A -85,B 0,C 180,E1 -22756.289,E2 -22756.289} C_VEL
LIN {X 0,Y 177.069,Z 775.349,A -85,B 0,C 180,E1 -22758.554,E2 -22758.554} C_VEL
LIN {X 0,Y 176.251,Z 776.42,A -85,B 0,C 180,E1 -22762.171,E2 -22762.171} C_VEL
LIN {X 0,Y 175.401,Z 776.675,A -85,B 0,C 180,E1 -22764.07,E2 -22764.07} C_VEL
LIN {X 0,Y 172.463,Z 776.763,A -85,B 0,C 180,E1 -22767.183,E2 -22767.183} C_VEL
LIN {X 0,Y 169.243,Z 777.025,A -85,B 0,C 180,E1 -22771.057,E2 -22771.057} C_VEL
LIN {X 0,Y 168.907,Z 777.294,A -85,B 0,C 180,E1 -22772.398,E2 -22772.398} C_VEL
LIN {X 0,Y 168.931,Z 777.729,A -85,B 0,C 180,E1 -22774.774,E2 -22774.774} C_VEL
LIN {X 0,Y 169.483,Z 777.395,A -85,B 0,C 180,E1 -22779.549,E2 -22779.549} C_VEL
LIN {X 0,Y 170.993,Z 775.572,A -85,B 0,C 180,E1 -22784.278,E2 -22784.278} C_VEL
LIN {X 0,Y 172.11,Z 774.07,A -85,B 0,C 180,E1 -22786.61,E2 -22786.61} C_VEL
LIN {X 0,Y 175.46,Z 769.832,A -85,B 0,C 180,E1 -22791.131,E2 -22791.131} C_VEL
LIN {X 0,Y 178.652,Z 765.507,A -85,B 0,C 180,E1 -22794.398,E2 -22794.398} C_VEL
LIN {X 0,Y 182.168,Z 760.101,A -85,B 0,C 180,E1 -22797.579,E2 -22797.579} C_VEL
LIN {X 0,Y 186.457,Z 753.452,A -85,B 0,C 180,E1 -22800.588,E2 -22800.588} C_VEL
LIN {X 0,Y 191.323,Z 745.34,A -85,B 0,C 180,E1 -22803.437,E2 -22803.437} C_VEL
LIN {X 0,Y 192.86,Z 742.257,A -85,B 0,C 180,E1 -22804.392,E2 -22804.392} C_VEL
LIN {X 0,Y 194.933,Z 734.711,A -85,B 0,C 180,E1 -22806.904,E2 -22806.904} C_VEL
LIN {X 0,Y 196.103,Z 726.826,A -85,B 0,C 180,E1 -22809.505,E2 -22809.505} C_VEL
LIN {X 0,Y 196.489,Z 719.569,A -85,B 0,C 180,E1 -22811.922,E2 -22811.922} C_VEL
LIN {X 0,Y 196.048,Z 713.354,A -85,B 0,C 180,E1 -22814.195,E2 -22814.195} C_VEL
LIN {X 0,Y 194.355,Z 706.758,A -85,B 0,C 180,E1 -22817.2,E2 -22817.2} C_VEL
LIN {X 0,Y 192.57,Z 701.618,A -85,B 0,C 180,E1 -22820.034,E2 -22820.034} C_VEL
LIN {X 0,Y 189.967,Z 695.013,A -85,B 0,C 180,E1 -22824.481,E2 -22824.481} C_VEL
LIN {X 0,Y 187.266,Z 688.918,A -85,B 0,C 180,E1 -22830.798,E2 -22830.798} C_VEL
LIN {X 0,Y 186.151,Z 687.194,A -85,B 0,C 180,E1 -22835.462,E2 -22835.462} C_VEL
LIN {X 0,Y 186.278,Z 686.767,A -85,B 0,C 180,E1 -22840.6,E2 -22840.6} C_VEL
LIN {X 0,Y 187.524,Z 687.354,A -85,B 0,C 180,E1 -22844.791,E2 -22844.791} C_VEL
LIN {X 0,Y 188.121,Z 689.304,A -85,B 0,C 180,E1 -22847.047,E2 -22847.047} C_VEL
LIN {X 0,Y 190.569,Z 692.741,A -85,B 0,C 180,E1 -22851.517,E2 -22851.517} C_VEL
LIN {X 0,Y 192.452,Z 696.333,A -85,B 0,C 180,E1 -22854.54,E2 -22854.54} C_VEL
LIN {X 0,Y 194.189,Z 700.008,A -85,B 0,C 180,E1 -22857.041,E2 -22857.041} C_VEL
LIN {X 0,Y 195.964,Z 705.46,A -85,B 0,C 180,E1 -22860,E2 -22860} C_VEL
LIN {X 0,Y 197.22,Z 710.901,A -85,B 0,C 180,E1 -22862.553,E2 -22862.553} C_VEL
LIN {X 0,Y 197.731,Z 718.71,A -85,B 0,C 180,E1 -22865.603,E2 -22865.603} C_VEL
LIN {X 0,Y 197.39,Z 725.957,A -85,B 0,C 180,E1 -22868.318,E2 -22868.318} C_VEL
LIN {X 0,Y 196.836,Z 729.924,A -85,B 0,C 180,E1 -22869.765,E2 -22869.765} C_VEL
LIN {X 0,Y 194.83,Z 734.114,A -85,B 0,C 180,E1 -22870.96,E2 -22870.96} C_VEL
LIN {X 0,Y 189.454,Z 743.392,A -85,B 0,C 180,E1 -22874.026,E2 -22874.026} C_VEL
LIN {X 0,Y 185.021,Z 750.13,A -85,B 0,C 180,E1 -22876.902,E2 -22876.902} C_VEL
LIN {X 0,Y 180.297,Z 756.78,A -85,B 0,C 180,E1 -22880.686,E2 -22880.686} C_VEL
LIN {X 0,Y 176.944,Z 761.065,A -85,B 0,C 180,E1 -22884,E2 -22884} C_VEL
LIN {X 0,Y 174.187,Z 764.29,A -85,B 0,C 180,E1 -22887.42,E2 -22887.42} C_VEL
LIN {X 0,Y 172.02,Z 766.534,A -85,B 0,C 180,E1 -22890.909,E2 -22890.909} C_VEL
LIN {X 0,Y 170.126,Z 768.027,A -85,B 0,C 180,E1 -22895.335,E2 -22895.335} C_VEL
LIN {X 0,Y 169.224,Z 768.293,A -85,B 0,C 180,E1 -22898.533,E2 -22898.533} C_VEL
LIN {X 0,Y 168.701,Z 767.8,A -85,B 0,C 180,E1 -22901.802,E2 -22901.802} C_VEL
LIN {X 0,Y 168.524,Z 766.55,A -85,B 0,C 180,E1 -22905.15,E2 -22905.15} C_VEL
LIN {X 0,Y 168.713,Z 764.466,A -85,B 0,C 180,E1 -22908.575,E2 -22908.575} C_VEL
LIN {X 0,Y 169.237,Z 761.4,A -85,B 0,C 180,E1 -22912.095,E2 -22912.095} C_VEL
LIN {X 0,Y 170.094,Z 757.133,A -85,B 0,C 180,E1 -22915.728,E2 -22915.728} C_VEL
LIN {X 0,Y 171.359,Z 751.403,A -85,B 0,C 180,E1 -22919.461,E2 -22919.461} C_VEL
LIN {X 0,Y 173.246,Z 744.063,A -85,B 0,C 180,E1 -22923.186,E2 -22923.186} C_VEL
LIN {X 0,Y 175.405,Z 736.078,A -85,B 0,C 180,E1 -22926.379,E2 -22926.379} C_VEL
LIN {X 0,Y 178.011,Z 726.121,A -85,B 0,C 180,E1 -22929.519,E2 -22929.519} C_VEL
LIN {X 0,Y 180.667,Z 715.508,A -85,B 0,C 180,E1 -22932.16,E2 -22932.16} C_VEL
LIN {X 0,Y 181.208,Z 712.546,A -85,B 0,C 180,E1 -22932.798,E2 -22932.798} C_VEL
LIN {X 0,Y 180,Z 701.391,A -85,B 0,C 180,E1 -22935.297,E2 -22935.297} C_VEL
LIN {X 0,Y 178.216,Z 690.221,A -85,B 0,C 180,E1 -22937.439,E2 -22937.439} C_VEL
LIN {X 0,Y 175.749,Z 678.671,A -85,B 0,C 180,E1 -22939.342,E2 -22939.342} C_VEL
LIN {X 0,Y 172.094,Z 665.079,A -85,B 0,C 180,E1 -22941.264,E2 -22941.264} C_VEL
LIN {X 0,Y 171.796,Z 663.263,A -85,B 0,C 180,E1 -22941.471,E2 -22941.471} C_VEL
LIN {X 0,Y 171.876,Z 663.071,A -85,B 0,C 180,E1 -22942.953,E2 -22942.953} C_VEL
LIN {X 0,Y 172.101,Z 663.042,A -85,B 0,C 180,E1 -22947.659,E2 -22947.659} C_VEL
LIN {X 0,Y 172.335,Z 663.018,A -85,B 0,C 180,E1 -22949.999,E2 -22949.999} C_VEL
LIN {X 0,Y 171.778,Z 663.086,A -85,B 0,C 180,E1 -22954.693,E2 -22954.693} C_VEL
LIN {X 0,Y 171.707,Z 663.089,A -85,B 0,C 180,E1 -22957.717,E2 -22957.717} C_VEL
LIN {X 0,Y 172.727,Z 665.977,A -85,B 0,C 180,E1 -22958.149,E2 -22958.149} C_VEL
LIN {X 0,Y 174.672,Z 671.678,A -85,B 0,C 180,E1 -22958.969,E2 -22958.969} C_VEL
LIN {X 0,Y 177.399,Z 684.311,A -85,B 0,C 180,E1 -22960.844,E2 -22960.844} C_VEL
LIN {X 0,Y 179.26,Z 695.175,A -85,B 0,C 180,E1 -22962.739,E2 -22962.739} C_VEL
LIN {X 0,Y 180.608,Z 706.008,A -85,B 0,C 180,E1 -22964.938,E2 -22964.938} C_VEL
LIN {X 0,Y 181.168,Z 712.099,A -85,B 0,C 180,E1 -22966.334,E2 -22966.334} C_VEL
LIN {X 0,Y 178.818,Z 722.158,A -85,B 0,C 180,E1 -22968.665,E2 -22968.665} C_VEL
LIN {X 0,Y 176.213,Z 732.317,A -85,B 0,C 180,E1 -22971.614,E2 -22971.614} C_VEL
LIN {X 0,Y 174.126,Z 740.095,A -85,B 0,C 180,E1 -22974.437,E2 -22974.437} C_VEL
LIN {X 0,Y 172.056,Z 747.919,A -85,B 0,C 180,E1 -22978.016,E2 -22978.016} C_VEL
LIN {X 0,Y 170.694,Z 753.623,A -85,B 0,C 180,E1 -22981.305,E2 -22981.305} C_VEL
LIN {X 0,Y 169.43,Z 759.252,A -85,B 0,C 180,E1 -22985.5,E2 -22985.5} C_VEL
LIN {X 0,Y 168.796,Z 762.387,A -85,B 0,C 180,E1 -22988.647,E2 -22988.647} C_VEL
LIN {X 0,Y 168.434,Z 764.8,A -85,B 0,C 180,E1 -22991.881,E2 -22991.881} C_VEL
LIN {X 0,Y 168.445,Z 766.482,A -85,B 0,C 180,E1 -22995.175,E2 -22995.175} C_VEL
LIN {X 0,Y 168.785,Z 767.421,A -85,B 0,C 180,E1 -22998.545,E2 -22998.545} C_VEL
LIN {X 0,Y 169.487,Z 767.546,A -85,B 0,C 180,E1 -23001.984,E2 -23001.984} C_VEL
LIN {X 0,Y 170.682,Z 766.848,A -85,B 0,C 180,E1 -23005.436,E2 -23005.436} C_VEL
LIN {X 0,Y 172.383,Z 765.299,A -85,B 0,C 180,E1 -23008.886,E2 -23008.886} C_VEL
LIN {X 0,Y 174.588,Z 762.838,A -85,B 0,C 180,E1 -23012.323,E2 -23012.323} C_VEL
LIN {X 0,Y 178.481,Z 757.995,A -85,B 0,C 180,E1 -23016.811,E2 -23016.811} C_VEL
LIN {X 0,Y 182.405,Z 752.584,A -85,B 0,C 180,E1 -23020.283,E2 -23020.283} C_VEL
LIN {X 0,Y 186.949,Z 745.684,A -85,B 0,C 180,E1 -23023.623,E2 -23023.623} C_VEL
LIN {X 0,Y 191.149,Z 738.747,A -85,B 0,C 180,E1 -23026.222,E2 -23026.222} C_VEL
LIN {X 0,Y 195.981,Z 729.878,A -85,B 0,C 180,E1 -23028.82,E2 -23028.82} C_VEL
LIN {X 0,Y 196.806,Z 727.047,A -85,B 0,C 180,E1 -23029.714,E2 -23029.714} C_VEL
LIN {X 0,Y 197.655,Z 719.474,A -85,B 0,C 180,E1 -23032.337,E2 -23032.337} C_VEL
LIN {X 0,Y 197.645,Z 710.865,A -85,B 0,C 180,E1 -23035.36,E2 -23035.36} C_VEL
LIN {X 0,Y 197.014,Z 706.187,A -85,B 0,C 180,E1 -23037.206,E2 -23037.206} C_VEL
LIN {X 0,Y 194.944,Z 699.09,A -85,B 0,C 180,E1 -23040.565,E2 -23040.565} C_VEL
LIN {X 0,Y 193.235,Z 694.334,A -85,B 0,C 180,E1 -23043.127,E2 -23043.127} C_VEL
LIN {X 0,Y 191.761,Z 691.641,A -85,B 0,C 180,E1 -23045.065,E2 -23045.065} C_VEL
LIN {X 0,Y 190.228,Z 688.461,A -85,B 0,C 180,E1 -23047.43,E2 -23047.43} C_VEL
LIN {X 0,Y 187.282,Z 683.113,A -85,B 0,C 180,E1 -23053.012,E2 -23053.012} C_VEL
LIN {X 0,Y 185.389,Z 681.472,A -85,B 0,C 180,E1 -23058.61,E2 -23058.61} C_VEL
LIN {X 0,Y 185.176,Z 681.407,A -85,B 0,C 180,E1 -23063.485,E2 -23063.485} C_VEL
LIN {X 0,Y 185.848,Z 682.288,A -85,B 0,C 180,E1 -23066.987,E2 -23066.987} C_VEL
LIN {X 0,Y 187.074,Z 683.763,A -85,B 0,C 180,E1 -23070.226,E2 -23070.226} C_VEL
LIN {X 0,Y 187.69,Z 684.772,A -85,B 0,C 180,E1 -23071.616,E2 -23071.616} C_VEL
LIN {X 0,Y 190.412,Z 689.542,A -85,B 0,C 180,E1 -23076.196,E2 -23076.196} C_VEL
LIN {X 0,Y 192.907,Z 694.462,A -85,B 0,C 180,E1 -23079.612,E2 -23079.612} C_VEL
LIN {X 0,Y 195.408,Z 701.259,A -85,B 0,C 180,E1 -23083.106,E2 -23083.106} C_VEL
LIN {X 0,Y 196.632,Z 705.323,A -85,B 0,C 180,E1 -23084.892,E2 -23084.892} C_VEL
LIN {X 0,Y 197.04,Z 709.869,A -85,B 0,C 180,E1 -23086.418,E2 -23086.418} C_VEL
LIN {X 0,Y 196.705,Z 718.882,A -85,B 0,C 180,E1 -23089.097,E2 -23089.097} C_VEL
LIN {X 0,Y 195.579,Z 727.645,A -85,B 0,C 180,E1 -23091.695,E2 -23091.695} C_VEL
LIN {X 0,Y 193.575,Z 736.635,A -85,B 0,C 180,E1 -23094.487,E2 -23094.487} C_VEL
LIN {X 0,Y 191.272,Z 743.003,A -85,B 0,C 180,E1 -23096.555,E2 -23096.555} C_VEL
LIN {X 0,Y 186.466,Z 751.44,A -85,B 0,C 180,E1 -23099.416,E2 -23099.416} C_VEL
LIN {X 0,Y 182.111,Z 758.304,A -85,B 0,C 180,E1 -23102.414,E2 -23102.414} C_VEL
LIN {X 0,Y 178.496,Z 763.838,A -85,B 0,C 180,E1 -23105.581,E2 -23105.581} C_VEL
LIN {X 0,Y 175.41,Z 768.275,A -85,B 0,C 180,E1 -23108.864,E2 -23108.864} C_VEL
LIN {X 0,Y 172.071,Z 772.599,A -85,B 0,C 180,E1 -23113.388,E2 -23113.388} C_VEL
LIN {X 0,Y 170.97,Z 774.161,A -85,B 0,C 180,E1 -23115.722,E2 -23115.722} C_VEL
LIN {X 0,Y 169.466,Z 776.048,A -85,B 0,C 180,E1 -23120.452,E2 -23120.452} C_VEL
LIN {X 0,Y 168.94,Z 776.426,A -85,B 0,C 180,E1 -23125.228,E2 -23125.228} C_VEL
LIN {X 0,Y 168.99,Z 775.889,A -85,B 0,C 180,E1 -23128.776,E2 -23128.776} C_VEL
LIN {X 0,Y 169.099,Z 776.46,A -85,B 0,C 180,E1 -23130.001,E2 -23130.001} C_VEL
LIN {X 0,Y 168.907,Z 777.294,A -85,B 0,C 180,E1 -23132.398,E2 -23132.398} C_VEL
LIN {X 0,Y 168.231,Z 777.664,A -85,B 0,C 180,E1 -23134.388,E2 -23134.388} C_VEL
LIN {X 0,Y 165.617,Z 777.71,A -85,B 0,C 180,E1 -23137.672,E2 -23137.672} C_VEL
LIN {X 0,Y 163.687,Z 777.241,A -85,B 0,C 180,E1 -23140.364,E2 -23140.364} C_VEL
LIN {X 0,Y 163.227,Z 776.607,A -85,B 0,C 180,E1 -23142.428,E2 -23142.428} C_VEL
LIN {X 0,Y 163.38,Z 776.322,A -85,B 0,C 180,E1 -23143.114,E2 -23143.114} C_VEL
LIN {X 0,Y 165.296,Z 774.173,A -85,B 0,C 180,E1 -23147.316,E2 -23147.316} C_VEL
LIN {X 0,Y 167.868,Z 771.279,A -85,B 0,C 180,E1 -23150.847,E2 -23150.847} C_VEL
LIN {X 0,Y 171.054,Z 767.426,A -85,B 0,C 180,E1 -23154.26,E2 -23154.26} C_VEL
LIN {X 0,Y 175.003,Z 762.006,A -85,B 0,C 180,E1 -23157.932,E2 -23157.932} C_VEL
LIN {X 0,Y 179.66,Z 755.472,A -85,B 0,C 180,E1 -23161.22,E2 -23161.22} C_VEL
LIN {X 0,Y 184.629,Z 747.815,A -85,B 0,C 180,E1 -23164.158,E2 -23164.158} C_VEL
LIN {X 0,Y 187.077,Z 743.409,A -85,B 0,C 180,E1 -23165.613,E2 -23165.613} C_VEL
LIN {X 0,Y 189.294,Z 736.339,A -85,B 0,C 180,E1 -23168.155,E2 -23168.155} C_VEL
LIN {X 0,Y 190.72,Z 728.706,A -85,B 0,C 180,E1 -23170.851,E2 -23170.851} C_VEL
LIN {X 0,Y 191.273,Z 721.797,A -85,B 0,C 180,E1 -23173.346,E2 -23173.346} C_VEL
LIN {X 0,Y 191.138,Z 717.777,A -85,B 0,C 180,E1 -23174.965,E2 -23174.965} C_VEL
LIN {X 0,Y 189.804,Z 711.228,A -85,B 0,C 180,E1 -23178.203,E2 -23178.203} C_VEL
LIN {X 0,Y 188.023,Z 705.466,A -85,B 0,C 180,E1 -23181.717,E2 -23181.717} C_VEL
LIN {X 0,Y 186.662,Z 701.475,A -85,B 0,C 180,E1 -23184.649,E2 -23184.649} C_VEL
LIN {X 0,Y 184.396,Z 695.304,A -85,B 0,C 180,E1 -23191.238,E2 -23191.238} C_VEL
LIN {X 0,Y 183.544,Z 693.895,A -85,B 0,C 180,E1 -23195.09,E2 -23195.09} C_VEL
LIN {X 0,Y 183.528,Z 693.341,A -85,B 0,C 180,E1 -23199.84,E2 -23199.84} C_VEL
LIN {X 0,Y 184.715,Z 693.88,A -85,B 0,C 180,E1 -23204.554,E2 -23204.554} C_VEL
LIN {X 0,Y 185.166,Z 695.725,A -85,B 0,C 180,E1 -23206.836,E2 -23206.836} C_VEL
LIN {X 0,Y 186.151,Z 697.23,A -85,B 0,C 180,E1 -23209.119,E2 -23209.119} C_VEL
LIN {X 0,Y 187.265,Z 699.169,A -85,B 0,C 180,E1 -23211.366,E2 -23211.366} C_VEL
LIN {X 0,Y 188.896,Z 702.629,A -85,B 0,C 180,E1 -23214.437,E2 -23214.437} C_VEL
LIN {X 0,Y 190.285,Z 706.282,A -85,B 0,C 180,E1 -23216.98,E2 -23216.98} C_VEL
LIN {X 0,Y 191.862,Z 712.631,A -85,B 0,C 180,E1 -23220.525,E2 -23220.525} C_VEL
LIN {X 0,Y 192.351,Z 717.126,A -85,B 0,C 180,E1 -23222.618,E2 -23222.618} C_VEL
LIN {X 0,Y 192.167,Z 724.723,A -85,B 0,C 180,E1 -23225.766,E2 -23225.766} C_VEL
LIN {X 0,Y 191.19,Z 731.468,A -85,B 0,C 180,E1 -23228.455,E2 -23228.455} C_VEL
LIN {X 0,Y 190.665,Z 733.024,A -85,B 0,C 180,E1 -23229.013,E2 -23229.013} C_VEL
LIN {X 0,Y 185.687,Z 741.388,A -85,B 0,C 180,E1 -23231.638,E2 -23231.638} C_VEL
LIN {X 0,Y 180.1,Z 749.574,A -85,B 0,C 180,E1 -23235.01,E2 -23235.01} C_VEL
LIN {X 0,Y 175.119,Z 756.212,A -85,B 0,C 180,E1 -23238.727,E2 -23238.727} C_VEL
LIN {X 0,Y 170.65,Z 761.469,A -85,B 0,C 180,E1 -23242.859,E2 -23242.859} C_VEL
LIN {X 0,Y 166.794,Z 765.518,A -85,B 0,C 180,E1 -23247.613,E2 -23247.613} C_VEL
LIN {X 0,Y 164.603,Z 767.422,A -85,B 0,C 180,E1 -23251.357,E2 -23251.357} C_VEL
LIN {X 0,Y 163.088,Z 768.356,A -85,B 0,C 180,E1 -23255.036,E2 -23255.036} C_VEL
LIN {X 0,Y 162.086,Z 768.44,A -85,B 0,C 180,E1 -23258.695,E2 -23258.695} C_VEL
LIN {X 0,Y 161.54,Z 767.72,A -85,B 0,C 180,E1 -23262.301,E2 -23262.301} C_VEL
LIN {X 0,Y 161.423,Z 766.223,A -85,B 0,C 180,E1 -23265.844,E2 -23265.844} C_VEL
LIN {X 0,Y 161.715,Z 763.924,A -85,B 0,C 180,E1 -23269.315,E2 -23269.315} C_VEL
LIN {X 0,Y 162.221,Z 760.901,A -85,B 0,C 180,E1 -23272.66,E2 -23272.66} C_VEL
LIN {X 0,Y 163.245,Z 756.072,A -85,B 0,C 180,E1 -23276.707,E2 -23276.707} C_VEL
LIN {X 0,Y 164.707,Z 749.987,A -85,B 0,C 180,E1 -23280.612,E2 -23280.612} C_VEL
LIN {X 0,Y 166.77,Z 742.334,A -85,B 0,C 180,E1 -23284.407,E2 -23284.407} C_VEL
LIN {X 0,Y 168.836,Z 734.839,A -85,B 0,C 180,E1 -23287.383,E2 -23287.383} C_VEL
LIN {X 0,Y 171.499,Z 725.115,A -85,B 0,C 180,E1 -23290.483,E2 -23290.483} C_VEL
LIN {X 0,Y 174.026,Z 715.256,A -85,B 0,C 180,E1 -23292.974,E2 -23292.974} C_VEL
LIN {X 0,Y 174.271,Z 712.567,A -85,B 0,C 180,E1 -23293.602,E2 -23293.602} C_VEL
LIN {X 0,Y 173.083,Z 701.368,A -85,B 0,C 180,E1 -23296.198,E2 -23296.198} C_VEL
LIN {X 0,Y 171.235,Z 690.021,A -85,B 0,C 180,E1 -23298.457,E2 -23298.457} C_VEL
LIN {X 0,Y 168.832,Z 678.735,A -85,B 0,C 180,E1 -23300.414,E2 -23300.414} C_VEL
LIN {X 0,Y 165.434,Z 666.017,A -85,B 0,C 180,E1 -23302.332,E2 -23302.332} C_VEL
LIN {X 0,Y 164.857,Z 663.945,A -85,B 0,C 180,E1 -23302.651,E2 -23302.651} C_VEL
LIN {X 0,Y 165.297,Z 663.895,A -85,B 0,C 180,E1 -23309.999,E2 -23309.999} C_VEL
LIN {X 0,Y 164.72,Z 663.967,A -85,B 0,C 180,E1 -23314.894,E2 -23314.894} C_VEL
LIN {X 0,Y 164.705,Z 663.966,A -85,B 0,C 180,E1 -23316.584,E2 -23316.584} C_VEL
LIN {X 0,Y 165.764,Z 666.892,A -85,B 0,C 180,E1 -23317.039,E2 -23317.039} C_VEL
LIN {X 0,Y 168.358,Z 673.802,A -85,B 0,C 180,E1 -23318.174,E2 -23318.174} C_VEL
LIN {X 0,Y 171.12,Z 687.368,A -85,B 0,C 180,E1 -23320.351,E2 -23320.351} C_VEL
LIN {X 0,Y 172.88,Z 698.8,A -85,B 0,C 180,E1 -23322.531,E2 -23322.531} C_VEL
LIN {X 0,Y 174.024,Z 709.576,A -85,B 0,C 180,E1 -23324.918,E2 -23324.918} C_VEL
LIN {X 0,Y 174.286,Z 713.156,A -85,B 0,C 180,E1 -23325.794,E2 -23325.794} C_VEL
LIN {X 0,Y 171.608,Z 723.911,A -85,B 0,C 180,E1 -23328.437,E2 -23328.437} C_VEL
LIN {X 0,Y 169.121,Z 733.225,A -85,B 0,C 180,E1 -23331.321,E2 -23331.321} C_VEL
LIN {X 0,Y 166.569,Z 742.42,A -85,B 0,C 180,E1 -23334.955,E2 -23334.955} C_VEL
LIN {X 0,Y 164.601,Z 749.792,A -85,B 0,C 180,E1 -23338.667,E2 -23338.667} C_VEL
LIN {X 0,Y 163.108,Z 755.811,A -85,B 0,C 180,E1 -23342.587,E2 -23342.587} C_VEL
LIN {X 0,Y 162.221,Z 759.888,A -85,B 0,C 180,E1 -23345.979,E2 -23345.979} C_VEL
LIN {X 0,Y 161.404,Z 764.071,A -85,B 0,C 180,E1 -23350.777,E2 -23350.777} C_VEL
LIN {X 0,Y 161.37,Z 766.745,A -85,B 0,C 180,E1 -23355.826,E2 -23355.826} C_VEL
LIN {X 0,Y 161.8,Z 767.654,A -85,B 0,C 180,E1 -23359.342,E2 -23359.342} C_VEL
LIN {X 0,Y 162.585,Z 767.76,A -85,B 0,C 180,E1 -23362.758,E2 -23362.758} C_VEL
LIN {X 0,Y 163.799,Z 767.152,A -85,B 0,C 180,E1 -23366.097,E2 -23366.097} C_VEL
LIN {X 0,Y 165.442,Z 765.872,A -85,B 0,C 180,E1 -23369.352,E2 -23369.352} C_VEL
LIN {X 0,Y 168.64,Z 762.617,A -85,B 0,C 180,E1 -23374.051,E2 -23374.051} C_VEL
LIN {X 0,Y 172.881,Z 757.696,A -85,B 0,C 180,E1 -23378.539,E2 -23378.539} C_VEL
LIN {X 0,Y 177.222,Z 752.099,A -85,B 0,C 180,E1 -23382.126,E2 -23382.126} C_VEL
LIN {X 0,Y 181.708,Z 745.713,A -85,B 0,C 180,E1 -23385.221,E2 -23385.221} C_VEL
